# B&R Automation Studio project TD52 (part 127)

#### MeNoiAL.h
```c
/********************************************************************
 * COPYRIGHT -- Bernecker + Rainer Industrie-Elektronik Ges.m.b.H.
 ********************************************************************
 * Program: MeNoiAL
 * File: MeNoiAL.h
 * Author: 120011115
 * Created: Mon Sep 05 16:14:57 2016
 ********************************************************************
 * Header for program MeNoiAL
 ********************************************************************
 * Generated with B&R Automation Studio Target for Simulink V4.2
 * (ERT based)
 ********************************************************************/

#ifndef RTW_HEADER_MeNoiAL_h_
#define RTW_HEADER_MeNoiAL_h_
#ifndef MeNoiAL_COMMON_INCLUDES_
# define MeNoiAL_COMMON_INCLUDES_
#include <math.h>
#include "rtwtypes.h"
#endif                                 /* MeNoiAL_COMMON_INCLUDES_ */

#include "MeNoiAL_types.h"
#include "lMeNoiAL.h"

/* Macros for accessing real-time model data structure */
#ifndef rtmGetErrorStatus
# define rtmGetErrorStatus(rtm)        ((void*) 0)
#endif

#ifndef rtmSetErrorStatus
# define rtmSetErrorStatus(rtm, val)   ((void) 0)
#endif

#ifndef rtmGetStopRequested
# define rtmGetStopRequested(rtm)      ((void*) 0)
#endif

#ifndef MIN
#define MIN(a,b)                       ((a) < (b) ? (a) : (b))
#endif

#ifndef MAX
#define MAX(a,b)                       ((a) > (b) ? (a) : (b))
#endif

/* user code (top of header file) */
/***************************************************************************************************
 * COPYRIGHT -- INNIO Jenbacher GmbH & CO OG
 ****************************************************************************************************
 * Program:            MeNoiAL
 * Author:             schmisi00
 * Created:            12.03.2020 09:42
 ****************************************************************************************************
 * MODEL INFORMATION
 ****************************************************************************************************
 * Model Name:         C:\Git\ValveFractureMonitoring\KN_MechNoiseAdapLim\MeNoiAL.slx
 * Model Version:      1.03
 * Simulink Version:   R2012b
 * B&R Target:         V4.5.1
 * Description:        Mechanical Noise Monitoring Function.
 *
 *                     Outstandings:
 *                     -------------
 *                     - NA
 ****************************************************************************************************
 * HISTORY
 ****************************************************************************************************
 * Last Modified By:   schmisi00
 * Last Modified Date: Thu Mar 12 09:41:58 2020
 * Modified Comment:   V1.00 - 20.09.2019 - Created, model implementation from AS to Simulink
 *                     V1.01 - 11.11.2019 - Removed trigger (Para.bMeNoi_Active) from adaptive limit calculation block
 *                     V1.02 - 21.11.2019 - Model cleanup, removed parameter rFiltGain_MeNoi and rFiltOffsFac_MeNoi
 *                     V1.03 - 12.03.2020 - Fenst2_Min calculation change to avoid 65535 during engine standstill
 ****************************************************************************************************/

/* Block signals (auto storage) */

/* Block states (auto storage) for system '<Root>' */

/* Invariant block signals (auto storage) */

/* External inputs (root inport signals with auto storage) */

/* External outputs (root outports fed by signals with auto storage) */

extern const ConstBlockIO_MeNoiAL MeNoiAL_ConstB;/* constant block i/o */

/* Model entry point functions */
extern void MeNoiAL_initialize(D_Work_MeNoiAL *MeNoiAL_DWork, struct fMeNoiAL* inst);
extern void MeNoiAL_step(BlockIO_MeNoiAL *MeNoiAL_B, D_Work_MeNoiAL
  *MeNoiAL_DWork, ExternalOutputs_MeNoiAL *MeNoiAL_Y, struct fMeNoiAL* inst);
extern void MeNoiAL_terminate(struct fMeNoiAL* inst);

/*-
 * The generated code includes comments that allow you to trace directly
 * back to the appropriate location in the model.  The basic format
 * is <system>/block_name, where system is the system number (uniquely
 * assigned by Simulink) and block_name is the name of the block.
 *
 * Use the MATLAB hilite_system command to trace the generated code back
 * to the model.  For example,
 *
 * hilite_system('<S3>')    - opens system 3
 * hilite_system('<S3>/Kp') - opens and selects block Kp which resides in S3
 *
 * Here is the system hierarchy for this model
 *
 * '<Root>' : 'MeNoiAL'
 * '<S1>'   : 'MeNoiAL/Environment Controller'
 * '<S2>'   : 'MeNoiAL/Environment Controller1'
 * '<S3>'   : 'MeNoiAL/Fenst2 Thresh Alarm'
 * '<S4>'   : 'MeNoiAL/Fenst2_Average_Min_Max'
 * '<S5>'   : 'MeNoiAL/Info'
 * '<S6>'   : 'MeNoiAL/Mechanical Noise Adaptive Limit'
 * '<S7>'   : 'MeNoiAL/PARA_Limitation'
 * '<S8>'   : 'MeNoiAL/Fenst2_Average_Min_Max/Divisor'
 * '<S9>'   : 'MeNoiAL/Fenst2_Average_Min_Max/MATLAB Function1'
 * '<S10>'  : 'MeNoiAL/Fenst2_Average_Min_Max/Divisor/Data Type Conversion Inherited'
 * '<S11>'  : 'MeNoiAL/Mechanical Noise Adaptive Limit/Backward Euler PT1'
 * '<S12>'  : 'MeNoiAL/Mechanical Noise Adaptive Limit/Divisor'
 * '<S13>'  : 'MeNoiAL/Mechanical Noise Adaptive Limit/Saturation Dynamic'
 * '<S14>'  : 'MeNoiAL/Mechanical Noise Adaptive Limit/Saturation Dynamic1'
 * '<S15>'  : 'MeNoiAL/Mechanical Noise Adaptive Limit/Backward Euler PT1/Divisor'
 * '<S16>'  : 'MeNoiAL/Mechanical Noise Adaptive Limit/Backward Euler PT1/Divisor/Data Type Conversion Inherited'
 * '<S17>'  : 'MeNoiAL/Mechanical Noise Adaptive Limit/Divisor/Data Type Conversion Inherited'
 */
#endif                                 /* RTW_HEADER_MeNoiAL_h_ */
```

#### MeNoiAL_private.h
```c
/********************************************************************
 * COPYRIGHT -- Bernecker + Rainer Industrie-Elektronik Ges.m.b.H.
 ********************************************************************
 * Program: MeNoiAL
 * File: MeNoiAL_private.h
 * Author: 120011115
 * Created: Mon Sep 05 16:14:57 2016
 ********************************************************************
 * Header for program MeNoiAL
 ********************************************************************
 * Generated with B&R Automation Studio Target for Simulink V4.2
 * (ERT based)
 ********************************************************************/

#ifndef RTW_HEADER_MeNoiAL_private_h_
#define RTW_HEADER_MeNoiAL_private_h_
#include "rtwtypes.h"
#include <bur/plctypes.h>
#ifndef __RTWTYPES_H__
#error This file requires rtwtypes.h to be included
#else
#ifdef TMWTYPES_PREVIOUSLY_INCLUDED
#error This file requires rtwtypes.h to be included before tmwtypes.h
#else

/* Check for inclusion of an incorrect version of rtwtypes.h */
#ifndef RTWTYPES_ID_C08S16I32L32N32F1
#error This code was generated with a different "rtwtypes.h" than the file included
#endif                                 /* RTWTYPES_ID_C08S16I32L32N32F1 */
#endif                                 /* TMWTYPES_PREVIOUSLY_INCLUDED */
#endif                                 /* __RTWTYPES_H__ */

#ifndef MIN
#define MIN(a,b)                       ((a) < (b) ? (a) : (b))
#endif

#ifndef MAX
#define MAX(a,b)                       ((a) > (b) ? (a) : (b))
#endif
#endif                                 /* RTW_HEADER_MeNoiAL_private_h_ */
```

#### MeNoiAL_types.h
```c
/********************************************************************
 * COPYRIGHT -- Bernecker + Rainer Industrie-Elektronik Ges.m.b.H.
 ********************************************************************
 * Program: MeNoiAL
 * File: MeNoiAL_types.h
 * Author: 120011115
 * Created: Mon Sep 05 16:14:57 2016
 ********************************************************************
 * Header for program MeNoiAL
 ********************************************************************
 * Generated with B&R Automation Studio Target for Simulink V4.2
 * (ERT based)
 ********************************************************************/

#ifndef RTW_HEADER_MeNoiAL_types_h_
#define RTW_HEADER_MeNoiAL_types_h_
#include "rtwtypes.h"
#ifndef MIN
#define MIN(a,b)                       ((a) < (b) ? (a) : (b))
#endif

#ifndef MAX
#define MAX(a,b)                       ((a) > (b) ? (a) : (b))
#endif

#endif                                 /* RTW_HEADER_MeNoiAL_types_h_ */
```

#### rtwtypes.h
```c
/********************************************************************
 * COPYRIGHT -- Bernecker + Rainer Industrie-Elektronik Ges.m.b.H.
 ********************************************************************
 * Program: MeNoiAL
 * File: rtwtypes.h
 * Author: 120011115
 * Created: Mon Sep 05 16:14:57 2016
 ********************************************************************
 * Header for program MeNoiAL
 ********************************************************************
 * Generated with B&R Automation Studio Target for Simulink V4.2
 * (ERT based)
 ********************************************************************/

#ifndef __RTWTYPES_H__
#define __RTWTYPES_H__
#ifndef TRUE
# define TRUE                          (1U)
#endif

#ifndef FALSE
# define FALSE                         (0U)
#endif

#ifndef __TMWTYPES__
#define __TMWTYPES__
#include <limits.h>

/*=======================================================================*
 * Target hardware information
 *   Device type: Intel->x86/Pentium
 *   Number of bits:     char:   8    short:   16    long:  32
 *                       long:  32
 *                       native word size:  32
 *   Byte ordering: LittleEndian
 *   Signed integer division rounds to: Zero
 *   Shift right on a signed integer as arithmetic shift: on
 *=======================================================================*/

/*=======================================================================*
 * Fixed width word size data types:                                     *
 *   int8_T, int16_T, int32_T     - signed 8, 16, or 32 bit integers     *
 *   uint8_T, uint16_T, uint32_T  - unsigned 8, 16, or 32 bit integers   *
 *   real32_T, real64_T           - 32 and 64 bit floating point numbers *
 *=======================================================================*/
typedef signed char int8_T;
typedef unsigned char uint8_T;
typedef short int16_T;
typedef unsigned short uint16_T;
typedef long int32_T;
typedef unsigned long uint32_T;
typedef float real32_T;
typedef double real64_T;

/*===========================================================================*
 * Generic type definitions: real_T, time_T, boolean_T, int_T, uint_T,       *
 *                           ulong_T, char_T and byte_T.                     *
 *===========================================================================*/
typedef double real_T;
typedef double time_T;
typedef unsigned char boolean_T;
typedef long int_T;
typedef unsigned long uint_T;
typedef unsigned long ulong_T;
typedef char char_T;
typedef unsigned char uchar_T;
typedef char_T byte_T;

/*=======================================================================*
 * Min and Max:                                                          *
 *   int8_T, int16_T, int32_T     - signed 8, 16, or 32 bit integers     *
 *   uint8_T, uint16_T, uint32_T  - unsigned 8, 16, or 32 bit integers   *
 *=======================================================================*/
#define MAX_int8_T                     ((int8_T)(127))
#define MIN_int8_T                     ((int8_T)(-128))
#define MAX_uint8_T                    ((uint8_T)(255U))
#define MIN_uint8_T                    ((uint8_T)(0U))
#define MAX_int16_T                    ((int16_T)(32767))
#define MIN_int16_T                    ((int16_T)(-32768))
#define MAX_uint16_T                   ((uint16_T)(65535U))
#define MIN_uint16_T                   ((uint16_T)(0U))
#define MAX_int32_T                    ((int32_T)(2147483647))
#define MIN_int32_T                    ((int32_T)(-2147483647-1))
#define MAX_uint32_T                   ((uint32_T)(0xFFFFFFFFU))
#define MIN_uint32_T                   ((uint32_T)(0U))

/* Logical type definitions */
#if (!defined(__cplusplus)) && (!defined(__true_false_are_keywords))
#  ifndef false
#   define false                       (0U)
#  endif

#  ifndef true
#   define true                        (1U)
#  endif
#endif

/*
 * Simulink Coder assumes the code is compiled on a target using a 2's complement representation
 * for signed integer values.
 */
#if ((SCHAR_MIN + 1) != -SCHAR_MAX)
#error "This code must be compiled using a 2's complement representation for signed integer values"
#endif

/* This ID is used to detect inclusion of an incompatible rtwtypes.h */
#define RTWTYPES_ID_C08S16I32L32N32F1
#else                                  /* __TMWTYPES__ */
#define TMWTYPES_PREVIOUSLY_INCLUDED
#endif                                 /* __TMWTYPES__ */

/* Block D-Work pointer type */
typedef void * pointer_T;

/* Simulink specific types */
#ifndef __SIMSTRUC_TYPES_H__
#define __SIMSTRUC_TYPES_H__

/* Trigger directions: falling, either, and rising */
typedef enum {
  FALLING_ZERO_CROSSING = -1,
  ANY_ZERO_CROSSING = 0,
  RISING_ZERO_CROSSING = 1
} ZCDirection;

/* Previous state of a trigger signal */
typedef uint8_T ZCSigState;

/* Initial value of a trigger zero crossing signal */
#define UNINITIALIZED_ZCSIG            0x03U
#define NEG_ZCSIG                      0x02U
#define POS_ZCSIG                      0x01U
#define ZERO_ZCSIG                     0x00U

/* Current state of a trigger signal */
typedef enum {
  FALLING_ZCEVENT = -1,
  NO_ZCEVENT = 0,
  RISING_ZCEVENT = 1
} ZCEventType;

#endif                                 /* __SIMSTRUC_TYPES_H__ */
#endif                                 /* __RTWTYPES_H__ */

#ifndef MIN
#define MIN(a,b)                       ((a) < (b) ? (a) : (b))
#endif

#ifndef MAX
#define MAX(a,b)                       ((a) > (b) ? (a) : (b))
#endif
```

#### MeNoiAL.c
```c
/********************************************************************
 * COPYRIGHT -- Bernecker + Rainer Industrie-Elektronik Ges.m.b.H.
 ********************************************************************
 * Program: MeNoiAL
 * File: MeNoiAL.c
 * Author: 120011115
 * Created: Mon Sep 05 16:14:57 2016
 ********************************************************************
 * Implementation of program MeNoiAL
 ********************************************************************
 * Generated with B&R Automation Studio Target for Simulink V4.2
 * (ERT based)
 ********************************************************************/
#include "MeNoiAL.h"
#include "MeNoiAL_private.h"

/*  Defines */

/*  Data Types */

/**************************** GLOBAL DATA *************************************/
/*  Definitions */

/*  Declarations  */

/***************************** FILE SCOPE DATA ********************************/

/*************************** FUNCTIONS ****************************************/

/* Model step function */
void MeNoiAL_step(struct BlockIO_MeNoiAL *MeNoiAL_B, struct D_Work_MeNoiAL *MeNoiAL_DWork,
                  ExternalOutputs_MeNoiAL *MeNoiAL_Y, struct fMeNoiAL* inst)
{
  /* local block i/o variables */
  boolean_T rtb_LogicalOperator;
  real32_T rtb_rFiltTau_MeNoi;
  real32_T rtb_rMargTExh_Active;
  real32_T rtb_rFenst2LiMn;
  real32_T rtb_Switch4;
  real32_T rtb_Divide;
  uint16_T rtb_Divide1[25];
  real32_T rtb_Switch;
  real32_T rtb_Switch3;
  real32_T rtb_Switch5;
  boolean_T rtb_y[25];
  real32_T rtb_Switch2_h[25];
  int32_T i;
  uint8_T rtb_SumofElements1;
  uint32_T tmp;
  boolean_T rtb_RelationalOperator_m;
  real32_T rtb_SumofElements_k;
  real32_T DiscreteTimeIntegrator[25];
  int32_T i_0;
  int32_T i_1;
  int16_T e_data[25];
  int16_T tmp_data[25];
  boolean_T rtb_LowerRelop;
  real32_T DiscreteTimeIntegrator_0;
  int32_T i_2;

  /* S-Function (bur_bus_in): '<Root>/Bus Input1' */
  MeNoiAL_B->BusInput1 = inst->Para;

  /* BusSelector: '<Root>/Bus Selector6' */
  rtb_rFiltTau_MeNoi = MeNoiAL_B->BusInput1.rFiltTau_MeNoi;
  rtb_rMargTExh_Active = MeNoiAL_B->BusInput1.rMargTExh_Active;
  rtb_rFenst2LiMn = MeNoiAL_B->BusInput1.rFenst2LiMn;

  /* Switch: '<S7>/Switch4' incorporates:
   *  BusSelector: '<Root>/Bus Selector6'
   *  Constant: '<S7>/Constant4'
   */
  if (MeNoiAL_B->BusInput1.rFenst2LiMx != 0.0F) {
    /* Saturate: '<S7>/Saturation4' */
    if (MeNoiAL_B->BusInput1.rFenst2LiMx >= 16000.0F) {
      rtb_Switch4 = 16000.0F;
    } else if (MeNoiAL_B->BusInput1.rFenst2LiMx <= 0.0F) {
      rtb_Switch4 = 0.0F;
    } else {
      rtb_Switch4 = MeNoiAL_B->BusInput1.rFenst2LiMx;
    }

    /* End of Saturate: '<S7>/Saturation4' */
  } else {
    rtb_Switch4 = 2000.0F;
  }

  /* End of Switch: '<S7>/Switch4' */

  /* S-Function (bur_bus_in): '<Root>/Bus Input' */
  MeNoiAL_B->BusInput = inst->In;

  /* Switch: '<S7>/Switch5' incorporates:
   *  Constant: '<S7>/Constant5'
   */
  if (rtb_rFenst2LiMn != 0.0F) {
    /* Saturate: '<S7>/Saturation5' */
    if (rtb_rFenst2LiMn >= 16000.0F) {
      rtb_Switch5 = 16000.0F;
    } else if (rtb_rFenst2LiMn <= 0.0F) {
      rtb_Switch5 = 0.0F;
    } else {
      rtb_Switch5 = rtb_rFenst2LiMn;
    }

    /* End of Saturate: '<S7>/Saturation5' */
  } else {
    rtb_Switch5 = 30.0F;
  }

  /* End of Switch: '<S7>/Switch5' */

  /* Switch: '<S7>/Switch' incorporates:
   *  Constant: '<S7>/Constant'
   */
  if (rtb_rFiltTau_MeNoi != 0.0F) {
    /* Saturate: '<S7>/Saturation' */
    if (rtb_rFiltTau_MeNoi >= 50.0F) {
      rtb_Switch = 50.0F;
    } else if (rtb_rFiltTau_MeNoi <= 0.0F) {
      rtb_Switch = 0.0F;
    } else {
      rtb_Switch = rtb_rFiltTau_MeNoi;
    }

    /* End of Saturate: '<S7>/Saturation' */
  } else {
    rtb_Switch = 5.0F;
  }

  /* End of Switch: '<S7>/Switch' */

  /* Product: '<S7>/Divide' incorporates:
   *  Constant: '<S7>/Constant2'
   */
  rtb_Divide = rtb_Switch4 / 3.5F;

  /* Switch: '<S7>/Switch3' incorporates:
   *  Constant: '<S7>/Constant3'
   */
  if (rtb_rMargTExh_Active != 0.0F) {
    /* Saturate: '<S7>/Saturation3' */
    if (rtb_rMargTExh_Active >= 1.0F) {
      rtb_Switch3 = 1.0F;
    } else if (rtb_rMargTExh_Active <= 0.0F) {
      rtb_Switch3 = 0.0F;
    } else {
      rtb_Switch3 = rtb_rMargTExh_Active;
    }

    /* End of Saturate: '<S7>/Saturation3' */
  } else {
    rtb_Switch3 = 0.15F;
  }

  /* End of Switch: '<S7>/Switch3' */

  /* Outputs for Atomic SubSystem: '<Root>/Fenst2_Average_Min_Max' */
  /* MATLAB Function: '<S4>/MATLAB Function1' */
  /* MATLAB Function 'Fenst2_Average_Min_Max/MATLAB Function1': '<S9>:1' */
  /* '<S9>:1:3' */
  for (i_0 = 0; i_0 < 25; i_0++) {
    rtb_y[i_0] = FALSE;
  }

  i_2 = (int32_T)((uint32_T)MeNoiAL_B->BusInput.ucNumCyl + 1U);
  if ((uint32_T)i_2 > 255U) {
    i_2 = 255;
  }

  if (2 > (uint8_T)i_2) {
    i = 1;
    i_2 = 0;
  } else {
    i = 2;
    i_2 = (uint8_T)i_2;
  }

  i_0 = i_2 - i;
  for (i_1 = 0; i_1 <= i_0; i_1++) {
    tmp_data[i_1] = (int16_T)(i + i_1);
  }

  i_0 = (i_2 - i) + 1;
  for (i_2 = 0; i_2 < i_0; i_2++) {
    for (i = 0; i < 1; i++) {
      e_data[i_2] = tmp_data[i_2];
    }
  }

  /* '<S9>:1:4' */
  for (i_2 = 0; i_2 < i_0; i_2++) {
    rtb_y[e_data[i_2] - 1] = TRUE;
  }

  /* output */
  /* '<S9>:1:7' */
  for (i_2 = 0; i_2 < 25; i_2++) {
    /* Logic: '<S4>/Logical Operator' incorporates:
     *  Logic: '<S4>/Logical Operator2'
     *  Product: '<S4>/Divide1'
     */
    rtb_RelationalOperator_m = (rtb_y[i_2] && (!MeNoiAL_B->
      BusInput.bKnockSig[i_2]));

    /* Product: '<S4>/Divide1' incorporates:
     *  DataTypeConversion: '<S4>/Data Type Conversion5'
     */
    rtb_Divide1[i_2] = (uint16_T)(rtb_RelationalOperator_m ?
      MeNoiAL_B->BusInput.uFenst2[i_2] : 0);

    /* Logic: '<S4>/Logical Operator' */
    rtb_y[i_2] = rtb_RelationalOperator_m;
  }

  /* End of MATLAB Function: '<S4>/MATLAB Function1' */

  /* Sum: '<S4>/Sum of Elements1' */
  tmp = (uint32_T)rtb_y[0];
  for (i_2 = 0; i_2 < 24; i_2++) {
    tmp += (uint32_T)rtb_y[i_2 + 1];
  }

  rtb_SumofElements1 = (uint8_T)tmp;

  /* End of Sum: '<S4>/Sum of Elements1' */

  /* Switch: '<S4>/Switch' incorporates:
   *  Constant: '<S4>/Constant2'
   *  DataTypeConversion: '<S4>/Data Type Conversion4'
   *  Product: '<S4>/Divide'
   */
  if (rtb_SumofElements1 != 0) {
    /* Sum: '<S4>/Sum of Elements' */
    rtb_SumofElements_k = (real32_T)rtb_Divide1[0];
    for (i_2 = 0; i_2 < 24; i_2++) {
      rtb_SumofElements_k += (real32_T)rtb_Divide1[i_2 + 1];
    }

    /* End of Sum: '<S4>/Sum of Elements' */

    /* Switch: '<S8>/Switch' incorporates:
     *  RelationalOperator: '<S8>/Relational Operator'
     */
    if (1 >= rtb_SumofElements1) {
      rtb_SumofElements1 = 1U;
    }

    /* End of Switch: '<S8>/Switch' */
    rtb_rFiltTau_MeNoi = rtb_SumofElements_k / (real32_T)rtb_SumofElements1;
  } else {
    rtb_rFiltTau_MeNoi = 0.0F;
  }

  /* End of Switch: '<S4>/Switch' */

  /* MinMax: '<S4>/MinMax1' */
  rtb_rMargTExh_Active = (real32_T)rtb_Divide1[0];
  for (i = 0; i < 24; i++) {
    if (!(rtb_rMargTExh_Active >= (real32_T)rtb_Divide1[i + 1])) {
      rtb_rMargTExh_Active = (real32_T)rtb_Divide1[i + 1];
    }
  }

  /* Switch: '<S4>/Switch2' incorporates:
   *  Constant: '<S4>/Constant3'
   */
  for (i_0 = 0; i_0 < 25; i_0++) {
    if (rtb_y[i_0]) {
      rtb_Switch2_h[i_0] = (real32_T)rtb_Divide1[i_0];
    } else {
      rtb_Switch2_h[i_0] = 65535.0F;
    }
  }

  /* End of Switch: '<S4>/Switch2' */

  /* MinMax: '<S4>/MinMax' */
  rtb_SumofElements_k = rtb_Switch2_h[0];
  for (i = 0; i < 24; i++) {
    if (!(rtb_SumofElements_k <= rtb_Switch2_h[i + 1])) {
      rtb_SumofElements_k = rtb_Switch2_h[i + 1];
    }
  }

  /* End of Outputs for SubSystem: '<Root>/Fenst2_Average_Min_Max' */

  /* Outputs for Atomic SubSystem: '<Root>/Mechanical Noise Adaptive Limit' */
  /* DataTypeConversion: '<S6>/Data Type Conversion1' */
  for (i_0 = 0; i_0 < 25; i_0++) {
    rtb_Switch2_h[i_0] = (real32_T)MeNoiAL_B->BusInput.uFenst2[i_0];
  }

  /* End of DataTypeConversion: '<S6>/Data Type Conversion1' */

  /* Outputs for Atomic SubSystem: '<S6>/Backward Euler PT1' */
  /* Switch: '<S15>/Switch' incorporates:
   *  Abs: '<S15>/Abs'
   *  RelationalOperator: '<S15>/Relational Operator'
   */
  if (2.22044605E-16F >= rtb_Switch) {
    rtb_rFenst2LiMn = 2.22044605E-16F;
  } else {
    rtb_rFenst2LiMn = rtb_Switch;
  }

  /* End of Switch: '<S15>/Switch' */

  /* RelationalOperator: '<S11>/Relational Operator' incorporates:
   *  Constant: '<S11>/Constant'
   */
  rtb_RelationalOperator_m = (rtb_Switch > 0.0F);

  /* Logic: '<S11>/Logical Operator' incorporates:
   *  Logic: '<S11>/Logical Operator1'
   */
  rtb_LogicalOperator = !rtb_RelationalOperator_m;

  /* DiscreteIntegrator: '<S11>/Discrete-Time Integrator' */
  if (MeNoiAL_DWork->DiscreteTimeIntegrator_IC_LOADI != 0) {
    for (i_0 = 0; i_0 < 25; i_0++) {
      MeNoiAL_DWork->DiscreteTimeIntegrator_DSTATE[i_0] = rtb_Switch2_h[i_0];
    }
  }

  /* Update for DiscreteIntegrator: '<S11>/Discrete-Time Integrator' */
  MeNoiAL_DWork->DiscreteTimeIntegrator_IC_LOADI = 0U;
  for (i_0 = 0; i_0 < 25; i_0++) {
    /* DiscreteIntegrator: '<S11>/Discrete-Time Integrator' incorporates:
     *  Delay: '<S11>/Delay'
     *  Product: '<S11>/Divide4'
     *  Sum: '<S11>/Sum4'
     */
    if (rtb_LogicalOperator || (MeNoiAL_DWork->DiscreteTimeIntegrator_PrevRese
         != 0)) {
      MeNoiAL_DWork->DiscreteTimeIntegrator_DSTATE[i_0] = rtb_Switch2_h[i_0];
    }

    DiscreteTimeIntegrator_0 = (rtb_Switch2_h[i_0] - MeNoiAL_DWork->
      Delay_DSTATE[i_0]) / rtb_rFenst2LiMn * 0.01F +
      MeNoiAL_DWork->DiscreteTimeIntegrator_DSTATE[i_0];

    /* Update for Delay: '<S11>/Delay' */
    MeNoiAL_DWork->Delay_DSTATE[i_0] = DiscreteTimeIntegrator_0;

    /* Update for DiscreteIntegrator: '<S11>/Discrete-Time Integrator' */
    MeNoiAL_DWork->DiscreteTimeIntegrator_DSTATE[i_0] = DiscreteTimeIntegrator_0;

    /* Sum: '<S6>/Add2' incorporates:
     *  Constant: '<S6>/Constant3'
     *  Product: '<S6>/Product1'
     *  Switch: '<S11>/Switch'
     */
    if (!rtb_RelationalOperator_m) {
      DiscreteTimeIntegrator_0 = rtb_Switch2_h[i_0];
    }

    DiscreteTimeIntegrator_0 = DiscreteTimeIntegrator_0 * 1.1F + rtb_Divide;

    /* End of Sum: '<S6>/Add2' */

    /* RelationalOperator: '<S13>/LowerRelop1' */
    rtb_LowerRelop = (DiscreteTimeIntegrator_0 > rtb_Switch4);

    /* Switch: '<S13>/Switch' incorporates:
     *  RelationalOperator: '<S13>/UpperRelop'
     */
    if (DiscreteTimeIntegrator_0 < rtb_Switch5) {
      DiscreteTimeIntegrator_0 = rtb_Switch5;
    }

    /* End of Switch: '<S13>/Switch' */

    /* Switch: '<S13>/Switch2' */
    if (rtb_LowerRelop) {
      DiscreteTimeIntegrator_0 = rtb_Switch4;
    }

    /* End of Switch: '<S13>/Switch2' */

    /* Product: '<S6>/Divide2' */
    DiscreteTimeIntegrator_0 = rtb_y[i_0] ? DiscreteTimeIntegrator_0 : 0.0F;
    DiscreteTimeIntegrator[i_0] = DiscreteTimeIntegrator_0;
  }

  /* Update for DiscreteIntegrator: '<S11>/Discrete-Time Integrator' */
  if (rtb_LogicalOperator) {
    MeNoiAL_DWork->DiscreteTimeIntegrator_PrevRese = 1;
  } else {
    MeNoiAL_DWork->DiscreteTimeIntegrator_PrevRese = 0;
  }

  /* End of Outputs for SubSystem: '<S6>/Backward Euler PT1' */

  /* Sum: '<S6>/Sum of Elements1' */
  tmp = (uint32_T)rtb_y[0];
  for (i_2 = 0; i_2 < 24; i_2++) {
    tmp += (uint32_T)rtb_y[i_2 + 1];
  }

  rtb_SumofElements1 = (uint8_T)tmp;

  /* End of Sum: '<S6>/Sum of Elements1' */

  /* Switch: '<S6>/Switch' incorporates:
   *  Constant: '<S6>/Constant2'
   *  DataTypeConversion: '<S6>/Data Type Conversion6'
   *  Product: '<S6>/Divide'
   */
  if (rtb_SumofElements1 != 0) {
    /* Sum: '<S6>/Sum of Elements' */
    rtb_rFenst2LiMn = DiscreteTimeIntegrator[0];
    for (i_2 = 0; i_2 < 24; i_2++) {
      rtb_rFenst2LiMn += DiscreteTimeIntegrator[i_2 + 1];
    }

    /* End of Sum: '<S6>/Sum of Elements' */

    /* Switch: '<S12>/Switch' incorporates:
     *  Constant: '<S12>/Constant2'
     *  RelationalOperator: '<S12>/Relational Operator'
     */
    if (1 >= rtb_SumofElements1) {
      i_2 = 1;
    } else {
      i_2 = rtb_SumofElements1;
    }

    /* End of Switch: '<S12>/Switch' */
    rtb_rFenst2LiMn /= (real32_T)i_2;
  } else {
    rtb_rFenst2LiMn = 0.0F;
  }

  /* End of Switch: '<S6>/Switch' */

  /* Sum: '<S6>/Add1' incorporates:
   *  Product: '<S6>/Product2'
   */
  rtb_rFenst2LiMn += rtb_Switch4 * rtb_Switch3;

  /* Switch: '<S14>/Switch2' incorporates:
   *  RelationalOperator: '<S14>/LowerRelop1'
   *  RelationalOperator: '<S14>/UpperRelop'
   *  Switch: '<S14>/Switch'
   */
  if (rtb_rFenst2LiMn > rtb_Switch4) {
    rtb_rFenst2LiMn = rtb_Switch4;
  } else {
    if (rtb_rFenst2LiMn < rtb_Switch5) {
      /* Switch: '<S14>/Switch' */
      rtb_rFenst2LiMn = rtb_Switch5;
    }
  }

  /* End of Switch: '<S14>/Switch2' */
  /* End of Outputs for SubSystem: '<Root>/Mechanical Noise Adaptive Limit' */

  /* Outputs for Atomic SubSystem: '<Root>/Fenst2 Thresh Alarm' */
  /* Switch: '<S3>/Switch' incorporates:
   *  Product: '<S3>/Product'
   */
  if (MeNoiAL_B->BusInput1.bMeNoi_Active) {
    for (i_0 = 0; i_0 < 25; i_0++) {
      rtb_Switch2_h[i_0] = DiscreteTimeIntegrator[i_0];
    }
  } else {
    for (i_0 = 0; i_0 < 25; i_0++) {
      rtb_Switch2_h[i_0] = rtb_Switch4 * MeNoiAL_ConstB.DataTypeConversion[i_0];
    }
  }

  for (i_0 = 0; i_0 < 25; i_0++) {
    /* RelationalOperator: '<S3>/Relational Operator' */
    rtb_LowerRelop = ((real32_T)rtb_Divide1[i_0] > rtb_Switch2_h[i_0]);

    /* Switch: '<S3>/Switch1' incorporates:
     *  Constant: '<S3>/Constant'
     *  Constant: '<S3>/Constant1'
     *  Delay: '<S3>/Delay'
     *  Sum: '<S3>/Sum'
     */
    if (rtb_LowerRelop) {
      rtb_SumofElements1 = (uint8_T)((uint32_T)MeNoiAL_DWork->Delay_DSTATE_c[i_0]
        + 1U);
    } else {
      rtb_SumofElements1 = 0U;
    }

    /* End of Switch: '<S3>/Switch1' */

    /* Logic: '<S3>/ 1' incorporates:
     *  Constant: '<S3>/Constant2'
     *  RelationalOperator: '<S3>/Relational Operator1'
     */
    rtb_RelationalOperator_m = ((rtb_SumofElements1 > 150) &&
      MeNoiAL_B->BusInput.bGCB_On_TC2_Di);

    /* Switch: '<S3>/Switch2' incorporates:
     *  Constant: '<S3>/Constant3'
     */
    if (rtb_RelationalOperator_m) {
      rtb_SumofElements1 = 150U;
    }

    /* End of Switch: '<S3>/Switch2' */

    /* Update for Delay: '<S3>/Delay' */
    MeNoiAL_DWork->Delay_DSTATE_c[i_0] = rtb_SumofElements1;

    /* BusCreator: '<Root>/Bus Creator' incorporates:
     *  Logic: '<S3>/ '
     *  Logic: '<S3>/ 2'
     *  Logic: '<S3>/Logical Operator'
     *  RelationalOperator: '<S3>/Relational Operator2'
     */
    MeNoiAL_Y->Out_MeNoiAL.bTExh_Mon_UseNarrowWindow[i_0] =
      ((MeNoiAL_B->BusInput1.bMeNoi_Active && rtb_LowerRelop) ||
       (MeNoiAL_B->BusInput1.bMeNoi_Active && (DiscreteTimeIntegrator[i_0] >
         rtb_rFenst2LiMn)));
    MeNoiAL_Y->Out_MeNoiAL.bValve[i_0] = rtb_RelationalOperator_m;

    /* BusCreator: '<Root>/Bus Creator1' */
    MeNoiAL_Y->Dbg_MeNoiAL.uMeNoi_Cnt[i_0] = rtb_SumofElements1;
    MeNoiAL_Y->Dbg_MeNoiAL.rFenst2_Vect[i_0] = (real32_T)rtb_Divide1[i_0];
    MeNoiAL_Y->Dbg_MeNoiAL.bValidCyl[i_0] = rtb_y[i_0];
  }

  /* End of Switch: '<S3>/Switch' */
  /* End of Outputs for SubSystem: '<Root>/Fenst2 Thresh Alarm' */

  /* Outputs for Atomic SubSystem: '<Root>/Fenst2_Average_Min_Max' */
  /* BusCreator: '<Root>/Bus Creator' incorporates:
   *  DataTypeConversion: '<S4>/Data Type Conversion1'
   *  DataTypeConversion: '<S4>/Data Type Conversion2'
   *  DataTypeConversion: '<S4>/Data Type Conversion3'
   *  MinMax: '<S4>/MinMax'
   *  MinMax: '<S4>/MinMax1'
   */
  MeNoiAL_Y->Out_MeNoiAL.uFenst2_Av = (uint16_T)(real32_T)fmod((real32_T)floor
    (rtb_rFiltTau_MeNoi), 65536.0F);
  MeNoiAL_Y->Out_MeNoiAL.uFenst2_Mx = (uint16_T)(int32_T)(real32_T)fmod
    (rtb_rMargTExh_Active, 65536.0F);
  MeNoiAL_Y->Out_MeNoiAL.uFenst2_Mn = (uint16_T)(int32_T)(real32_T)fmod
    (rtb_SumofElements_k, 65536.0F);

  /* End of Outputs for SubSystem: '<Root>/Fenst2_Average_Min_Max' */

  /* BusCreator: '<Root>/Bus Creator1' */
  MeNoiAL_Y->Dbg_MeNoiAL.rFiltTau_Lim = rtb_Switch;
  MeNoiAL_Y->Dbg_MeNoiAL.rFiltGain_Lim = 0.0F;
  MeNoiAL_Y->Dbg_MeNoiAL.rMargTexhAct_Lim = rtb_Switch3;
  MeNoiAL_Y->Dbg_MeNoiAL.rOffMeNoi_Lim = rtb_Divide;
  MeNoiAL_Y->Dbg_MeNoiAL.rFenst2LiMx_Lim = rtb_Switch4;
  MeNoiAL_Y->Dbg_MeNoiAL.rFenst2LiMn_Lim = rtb_Switch5;
  for (i_0 = 0; i_0 < 25; i_0++) {
    MeNoiAL_Y->Dbg_MeNoiAL.uAdapLim_MeNoi_Cyl[i_0] = DiscreteTimeIntegrator[i_0];
  }

  MeNoiAL_Y->Dbg_MeNoiAL.uAdapLim_Marg = rtb_rFenst2LiMn;

  /* S-Function (bur_bus_out): '<Root>/Bus Output' */
  inst->Out = MeNoiAL_Y->Out_MeNoiAL;

  /* S-Function (bur_bus_out): '<Root>/Bus Output1' */
  inst->Dbg = MeNoiAL_Y->Dbg_MeNoiAL;

  /* UnitDelay: '<S5>/Unit Delay' */
  MeNoiAL_B->UnitDelay = MeNoiAL_DWork->UnitDelay_DSTATE;

  /* S-Function (bur_out): '<Root>/Output' */
  inst->Version = MeNoiAL_B->UnitDelay;

  /* Update for UnitDelay: '<S5>/Unit Delay' */
  MeNoiAL_DWork->UnitDelay_DSTATE = 103U;
}

/* Model initialize function */
void MeNoiAL_initialize(struct D_Work_MeNoiAL *MeNoiAL_DWork, struct fMeNoiAL* inst)
{
  /* InitializeConditions for Atomic SubSystem: '<Root>/Mechanical Noise Adaptive Limit' */
  /* InitializeConditions for Atomic SubSystem: '<S6>/Backward Euler PT1' */
  /* InitializeConditions for DiscreteIntegrator: '<S11>/Discrete-Time Integrator' */
  MeNoiAL_DWork->DiscreteTimeIntegrator_IC_LOADI = 1U;

  /* End of InitializeConditions for SubSystem: '<S6>/Backward Euler PT1' */
  /* End of InitializeConditions for SubSystem: '<Root>/Mechanical Noise Adaptive Limit' */
}

/* Model terminate function */
void MeNoiAL_terminate(struct fMeNoiAL* inst)
{
  /* (no terminate code required) */
}

/*======================== TOOL VERSION INFORMATION ==========================*
 * MATLAB 8.0 (R2012b)20-Jul-2012                                             *
 * Simulink 8.0 (R2012b)20-Jul-2012                                           *
 * Simulink Coder 8.3 (R2012b)20-Jul-2012                                     *
 * Embedded Coder 6.3 (R2012b)20-Jul-2012                                     *
 * Stateflow 8.0 (R2012b)20-Jul-2012                                          *
 *============================================================================*/

/*======================= LICENSE IN USE INFORMATION =========================*
 * matlab                                                                     *
 * matlab_coder                                                               *
 * real-time_workshop                                                         *
 * rtw_embedded_coder                                                         *
 * simulink                                                                   *
 *============================================================================*/
```

#### MeNoiAL_data.c
```c
/********************************************************************
 * COPYRIGHT -- Bernecker + Rainer Industrie-Elektronik Ges.m.b.H.
 ********************************************************************
 * Program: MeNoiAL
 * File: MeNoiAL_data.c
 * Author: 120011115
 * Created: Mon Sep 05 16:14:57 2016
 ********************************************************************
 * Data for program MeNoiAL
 ********************************************************************
 * Generated with B&R Automation Studio Target for Simulink V4.2
 * (ERT based)
 ********************************************************************/
#include "MeNoiAL.h"
#include "MeNoiAL_private.h"

/*  GLOBAL DATA DEFINITIONS */

/* Invariant block signals (auto storage) */
const ConstBlockIO_MeNoiAL MeNoiAL_ConstB = {
  { 1.0F, 1.0F, 1.0F, 1.0F, 1.0F, 1.0F, 1.0F, 1.0F, 1.0F, 1.0F, 1.0F, 1.0F, 1.0F,
    1.0F, 1.0F, 1.0F, 1.0F, 1.0F, 1.0F, 1.0F, 1.0F, 1.0F, 1.0F, 1.0F, 1.0F }
  /* '<S3>/Data Type Conversion' */
};
```

#### fMeNoiAL.c
```c
/********************************************************************
 * COPYRIGHT -- Bernecker + Rainer Industrie-Elektronik Ges.m.b.H.
 ********************************************************************
 * Program: MeNoiAL
 * File: fMeNoiAL.c
 * Author: 120011115
 * Created: Mon Sep 05 16:14:57 2016
 ********************************************************************
 * Implementation of program MeNoiAL
 ********************************************************************
 * Generated with B&R Automation Studio Target for Simulink V4.2
 * (ERT based)
 ********************************************************************/
#include <bur/plctypes.h>
#include "MeNoiAL.h"
#include "rtwtypes.h"

/* Defines */
#define SS_TERMINATE 4
#define SS_OUTPUT 3
#define SS_INITIALIZE 2

/*  Data Types */

/**************************** GLOBAL DATA *************************************/
/*  Definitions */

/*  Declarations  */

/***************************** FILE SCOPE DATA ********************************/

/*************************** FUNCTIONS ****************************************/
#ifdef __cplusplus

unsigned long bur_heap_size = 6553500;

#endif

void fMeNoiAL(struct fMeNoiAL* inst)
{
  BlockIO_MeNoiAL *MeNoiAL_B = &(inst)->bur_BlockIO_MeNoiAL;
	D_Work_MeNoiAL *MeNoiAL_DWork = &(inst)->bur_D_Work_MeNoiAL;
	ExternalOutputs_MeNoiAL *MeNoiAL_Y = &(inst)->bur_ExternalOutputs_MeNoiAL;

  switch (inst->ssMethodType)
  {
   case SS_INITIALIZE:
    /* call model initialize function */
    MeNoiAL_initialize(MeNoiAL_DWork, inst);
    break;

   case SS_OUTPUT:
    /* call model step function */
    MeNoiAL_step(MeNoiAL_B, MeNoiAL_DWork, MeNoiAL_Y, inst);

    break;

   case SS_TERMINATE:
    /* call model terminate function */
    MeNoiAL_terminate(inst);
    break;
  }
}

/*****************************************************************************
   Function block sample time: 0.01s
 *****************************************************************************/

/*****************************************************************************
   B&R Automation Studio Target for Simulink Version: A4.5.1 (27-Jul-2015)
 *****************************************************************************/

/*======================== TOOL VERSION INFORMATION ==========================*
 * MATLAB 8.0 (R2012b)20-Jul-2012                                             *
 * Simulink 8.0 (R2012b)20-Jul-2012                                           *
 * Simulink Coder 8.3 (R2012b)20-Jul-2012                                     *
 * Embedded Coder 6.3 (R2012b)20-Jul-2012                                     *
 * Stateflow 8.0 (R2012b)20-Jul-2012                                          *
 *============================================================================*/

/*======================= LICENSE IN USE INFORMATION =========================*
 * matlab                                                                     *
 * matlab_coder                                                               *
 * real-time_workshop                                                         *
 * rtw_embedded_coder                                                         *
 * simulink                                                                   *
 *============================================================================*/
```

#### lib_properties.txt
```
For manual assignment to hardware configuration please
add the following additional include directories:

\Logical\MATLAB_includes\R2012b\

And the following additional build options:

-lm -D MODEL=MeNoiAL -D NUMST=1 -D NCSTATES=0 -D HAVESTDIO -D ONESTEPFCN=1 -D TERMFCN=1 -D MAT_FILE=0 -D MULTI_INSTANCE_CODE=1 -D INTEGER_CODE=0 -D MT=0 -D CLASSIC_INTERFACE=0 -D TID01EQ=0
```

### Data object Logical/Knocking/META_KN (Simple) - MODUL META data file

#### META_KN.dat
```
; *******************************************************************************
; AGGR: Module Meta Data (data module)
;
; This code is confidential and proprietary to the INNIO Company.
; It may not be used in any form, or reproduced in any manner, without the express
; written permission of the INNIO Company.
; Copyright, INNIO Company, 2025
;
; Customized modifications: -
; ------------------------
;
; History:
; -------
; V3.99			06-03-2013	Weitzer, 	generated for modular software
; V4.00 		31.01.2014	Weitzer, 	versions changed
; V4.01.00.00 	23.07.2014	Waldhart,	new interfaces added
; V4.02.00.00	16.02.2015	Caks,		added safi dmr
; V4.03.00.00	02.11.2015	Zengerer	add MANDATORYMODULE statement
; V4.04.00.00   18.04.2016	Gwiggner,   Bugfix ITP Interpolation GAS1-2
; V4.04.00.00	12.05.2016	502423184	versions changed,  SAFI_DMR Task for Type9 / G2
; V4.04.00.00	14.11.2016	Gwiggner	Bugfix: VISU knocking IP reduction
; V4.04.00.00   xx.03.2017	Farre,		Bugfix: adaptive knock limit safi_kls
; V4.04.00.00   15.05.2017	Gwiggner,	Bugfix: KLS98 validation - MSF not working
; V4.05.00.00   05.03.2018	Perktold,	Delaytime for MSF SAFI/KLS corrected 2.5sec instead of 0.3s, Type 6 "BlockAfterKnockTrip"
; V4.05.01.00   16.04.2018	Perktold,	Integrated comments regarding "Safety-related application software source code (EN 13849-1 / 4.6.3)"
; V4.06.00.00   28.09.2018	Gwiggner,	change A3342 Knock sensor measuring sensor failure from Prio 3 to Prio 2"
; V4.07.00.00	13.05.2019	Hohensinner	Added RKS Package
; V4.07.00.00	23.10.2019	Farre,		BU 01: avoiding division by 0
; V4.09.00.00	23.01.2020	Schmidt,	Mechanical noise monitoring for valve fracture detection added
; V4.10.00.00	19.01.2020	Farre,		added individual knocking threshold per Bank
; V4.10.00.00	28.01.2021	Denk,		Alarm deactivation when DGS/WinMOD Simulation is active (2438, 2439, 2440, 2441).
; V4.11.00.00	22.12.2021	Andre		Moved W2493 and B2939 to SAFI module. Added notification of frozen or knock noise from SAFI module.
; V4.11.00.00	14.01.2022	Schmidt		Changed bKnockSig variable to global (used for PU scuffing detection)
; V4.12.00.00	03.10.2022	Farre,		Issue #438: Current knock integrator value connected to AVG, MAX & MIN MM2VIS for KLS90
; 				03.10.2022	Farre,		Issue #906: J208 KLS90 uses only one knock sensor, second sensor is looped through
;				22.11.2022	Farre,		Feature: Introduction knock adaptive limit for Type4 with DMR
;				19.12.2022	Perktold	added comments for sr-code (EN 13849-1 / 4.6.3) for A3342
; V04.13.00.00	05.12.2023	Bencze		A1048,3339,3342: risc class 10 (for T6), no remote reset possible
; V04.14.00.00	19.07.2024	Kafka,		Remove G2 and add KLS as RKS system for T9
;							Andre,		Fix issue 1585.
;				21.01.2025	Gwiggner,	J208F KLS90 use of 2nd knock senor (#1791)
;
; Instructions for use:
; --------------------
; make only changes at the version numbers
;
; Outstandings:
; ------------
;
; *******************************************************************************
;
"<META>"
;
; Module ID
"<MODUL>KN</MODUL>"
;
; Module Version (xx.yy.zz.cc)
"<VERSION>04.14.00.00</VERSION>"
;
; Module Basisupdate Version BU (00-99)
"<BASISUPDATE_VERSION>00</BASISUPDATE_VERSION>"
;
; Optional: specify order number for limitated module usage
"<ORDER></ORDER>" ;<!--(optional for restricted customizations; missing statement makes module valid for all orders)-->
;
; Parameter Check <PARAn Name='aAbcdef' MIN='xxx' MAX='yyy' />  (watch for correct spacings and apostrophs!)
"<PARAMETER_CHK>"
"<PARA1 Name='iEng_Motortype' MIN='208' MAX='920' />"
"<PARA2 />"
"<PARA3 />"
"<PARA4 />"
"<PARA5 />"
"</PARAMETER_CHK>"
;
; Statement, that this module´s parameter check passing is mandatory (KN is allways mandatory, so other statements than TRUE here in this module are ignored)
"<MANDATORYMODULE>TRUE</MANDATORYMODULE>"
;
; Permanent Datamodule Filenames<!-- NAME ist ohne Dateiendung einzutragen; Nur für Counter und interne Parameter verwenden-->
"<DATAMODULES>" ;<!-- optional; mehrere DATAMODULES erlaubt-->
"	<DATAMODULE>par_KN</DATAMODULE>"
"</DATAMODULES>"
;
; Dependencies Modules (MMxx.yy.zz.cc)
"<DEPENDENCIES>"
"	<DEPENDENCY MODULE='SA' VERSION='04.14.00.00' />"
"	<DEPENDENCY MODULE='OP' VERSION='04.03.00.00' />"
"	<DEPENDENCY MODULE='AB' VERSION='04.03.00.00' />"
"	<DEPENDENCY MODULE='IG' VERSION='04.01.00.00' />"
"	<DEPENDENCY MODULE='KL' VERSION='04.03.00.00' />"
"	<DEPENDENCY MODULE='PB' VERSION='04.00.04.00' />"
"	<DEPENDENCY MODULE='VI' VERSION='04.00.00.00' />"
"	<DEPENDENCY MODULE='HA' VERSION='04.07.00.00' />"
"	<DEPENDENCY MODULE='EC' VERSION='04.14.00.00' />"
"	<DEPENDENCY MODULE='GT' VERSION='04.07.00.00' />"
"   <DEPENDENCY VISVERSION='02.15.00.00' />"			; Dependencies Visualization
"</DEPENDENCIES>"
;
; Module function description
"<MODULEFUNCTION>" ;<!-- short overview documentation of module function; add reference to detailed information, if available-->
"	<General>	"
"	Knocking Prevention "
"	</General>	"
""
"	<F1 Name='enter name of main function 1 here' LastModified='4.0.0.0'>"
"	o knocking monitoring with KLS90	"
"	</F1>"
"	<F3 Name='enter name of main function 2 here' LastModified='4.0.0.0'>"
"	o knocking monitoring with KLS98	"
"	</F2>"
"	<F3 Name='enter name of main function 3 here' LastModified='4.0.0.0'>"
"	o knocking monitoring with SAFIKLS	"
"	</F3>"
""
"	<Info>"
"	 V4.01.00.00	new interfaces added"
"	 V4.02.00.00	added safi dmr"
"	 V4.03.00.00	add MANDATORYMODULE statement"
"	 V4.04.00.00	versions changed"
" 	 V4.04.00.00	VISU knocking IP reduction"
"    V4.04.00.00    Bugfix: KLS98 validation - MSF not working "
"    V4.05.01.00    BU 01: change A3342 Knock sensor measuring sensor failure from Prio 3 to Prio 2"
" 	 V4.07.00.00	Added RKS package"
"	 V4.07.00.00	BU 01: avoiding division by 0"
"	<Customized LastModified='4.0.0.0'>	"
"	- Nothing "
"	</Customized>	"
""
"</MODULEFUNCTION>"
;
"</META>"
```

### module_Knocking.typ - Package data types
```iecst
(********************************************************************
 * COPYRIGHT -- INNIO Company
 ********************************************************************
 * Package: Knocking
 * File: module_Knocking.typ
 * Author: WaldharM
 * Created: October 03, 2011
 ********************************************************************
 * Data types of package Knocking
 ********************************************************************)

TYPE
	IN_KN_Struct : 	STRUCT  (* general*)
		tMS_PBC0 : ARRAY[0..12]OF _tSAFImdatas; (* Pressure based control measuring data 0*) (* OldName: DMR_md1; Cycle:2; *)
		tMS_PBC1 : ARRAY[0..12]OF _tSAFImdatas; (* Pressure based control measuring data 1 *) (* OldName: DMR_md1; Cycle:2; *)
		tMS_PBC2 : ARRAY[0..12]OF _tSAFImdatas; (* Pressure based control measuring data 2 *) (* OldName: DMR_md2; Cycle:2; *)
		tMS_PBC3 : ARRAY[0..12]OF _tSAFImdatas; (* Pressure based control measuring data 3 *) (* OldName: DMR_md3; Cycle:2; *)
		tMS_PBC4 : ARRAY[0..12]OF _tSAFImdatas; (* Pressure based control measuring data 4 *) (* OldName: DMR_md4; Cycle:2; *)
		tMS_PBC5 : ARRAY[0..12]OF _tSAFImdatas; (* Pressure based control measuring data 5 *) (* OldName: DMR_md5; Cycle:2; *)
		tMS_PBC6 : ARRAY[0..12]OF _tSAFImdatas; (* Pressure based control measuring data 6 *) (* OldName: DMR_md6; Cycle:2; *)
		tMS_PBC7 : ARRAY[0..12]OF _tSAFImdatas; (* Pressure based control measuring data 7 *) (* OldName: DMR_md7; Cycle:2; *)
		tMS_PBC8 : ARRAY[0..12]OF _tSAFImdatas; (* Pressure based control measuring data 8 *) (* OldName: DMR_md8; Cycle:2; *)
		tMS_PBC9 : ARRAY[0..12]OF _tSAFImdatas; (* Pressure based control measuring data 9 *) (* OldName: DMR_md9; Cycle:2; *)
		tMS_PBC10 : ARRAY[0..12]OF _tSAFImdatas; (* Pressure based control measuring data 10 *) (* OldName: DMR_md10; Cycle:2; *)
		tMS_PBC11 : ARRAY[0..12]OF _tSAFImdatas; (* Pressure based control measuring data 11 *) (* OldName: DMR_md11; Cycle:2; *)
		tMS_PBC12 : ARRAY[0..12]OF _tSAFImdatas; (* Pressure based control measuring data 12 *) (* OldName: DMR_md12; Cycle:2; *)
		tMS_PBC13 : ARRAY[0..12]OF _tSAFImdatas; (* Pressure based control measuring data 13 *) (* OldName: DMR_md13; Cycle:2; *)
		tMS_PBC14 : ARRAY[0..12]OF _tSAFImdatas; (* Pressure based control measuring data 14 *) (* OldName: DMR_md14; Cycle:2; *)
		tMS_PBC15 : ARRAY[0..12]OF _tSAFImdatas; (* Pressure based control measuring data 15 *) (* OldName: DMR_md15; Cycle:2; *)
		tMS_PBC16 : ARRAY[0..12]OF _tSAFImdatas; (* Pressure based control measuring data 16 *) (* OldName: DMR_md16; Cycle:2; *)
		tMS_PBC17 : ARRAY[0..12]OF _tSAFImdatas; (* Pressure based control measuring data 17 *) (* OldName: DMR_md17; Cycle:2; *)
		tMS_PBC18 : ARRAY[0..12]OF _tSAFImdatas; (* Pressure based control measuring data 18 *) (* OldName: DMR_md18; Cycle:2; *)
		tMS_PBC19 : ARRAY[0..12]OF _tSAFImdatas; (* Pressure based control measuring data 19 *) (* OldName: DMR_md19; Cycle:2; *)
		rP_Act_Norm_Filt : REAL; (* actual power related to rP_Nom filtered T=1s  [%/P_Nom] *) (* OldName: P_IST; Cycle:2; *)
		tAB2KN : AmmBase2MM; (* 0 *) (* OldName: 0; Cycle:2; *)
		rN_EngAct : REAL; (* engine speed *) (* OldName: n_ist; Cycle:2; *)
		iSt_OpMode : UDINT; (* engine operation mode *) (* OldName: 0; Cycle:2; *)
		tP_Act : ARRAY[0..2]OF HALioAi_Type; (* actual electric power [KW] *) (*OldName:ssPAct;Cycle:2;*)
		rP_Nom : REAL; (* nominal power *) (* OldName: 0; Cycle:2; *)
		rKLS98_X_Window1 : ARRAY[0..24]OF REAL; (* cylinder values of KLS98 window 1 *) (* OldName: Fenst1; Cycle:2; *)
		rKLS98_X_Window2 : ARRAY[0..24]OF REAL; (* cylinder values of KLS98 window 2 *) (* OldName: Fenst2; Cycle:2; *)
		rKLS98_X_Window3 : ARRAY[0..24]OF REAL; (* cylinder values of KLS98 window 3 *) (* OldName: Fenst3; Cycle:2; *)
		rKLS98_X_Window4 : ARRAY[0..24]OF REAL; (* cylinder values of KLS98 window 4 *) (* OldName: Fenst4; Cycle:2; *)
		tGCB_On_TC2 : HALioDi_Type; (* DI: Generator circuit breaker closed, TC2 synchron *) (* OldName: GCB_ON_TC1 ; Cycle:2; *)
		iU_SAFI_Win1 : ARRAY[0..24]OF INT; (* cylinder values of KLS window 1 *) (* OldName: Fenst1; Cycle:2; *)
		iU_SAFI_Win2 : ARRAY[0..24]OF INT; (* cylinder values of KLS window 2 *) (* OldName: Fenst2; Cycle:2; *)
		iU_SAFI_Win3 : ARRAY[0..24]OF INT; (* cylinder values of KLS window 3 *) (* OldName: Fenst3; Cycle:2; *)
		iU_SAFI_Win4 : ARRAY[0..24]OF INT; (* cylinder values of KLS window 4 *) (* OldName: Fenst4; Cycle:2; *)
		tPB2MM : ParaBase2MM_type; (* Messages from parametercheck module parameter are OK *) (* OldName: new PV; Cycle:2; *)
		tKLS90_1 : HALioAi_Type; (* AI: KLS90 sensor 1 signal *) (* OldName: ssKLS_Signal1; Cycle:2; *)
		tKLS90_2 : HALioAi_Type; (* AI: KLS90 sensor 1 signal *) (* OldName: ssKLS_Signal2; Cycle:2; *)
		tEng_Run : HALioDo_Type; (* engine operating state *) (* OldName: M_BTRB; Cycle:5; *)
		iIdx_OMSS : INT; (* index of operation mode selector switch *) (* OldName: BWS_HA; Cycle:2; *)
		iPassLevel : INT; (*pass level actual*) (*OldName:ucPassLevel; Cycle:5;*)
		bGasTyp1_Act : BOOL; (* gas type 1 active *) (*OldName:AN_GAS1,AW_ZZP1;Cycle:2;*)
		bGasTyp2_Act : BOOL; (* gas type 2 active *) (*OldName:AN_GAS2,AW_ZZP2;Cycle:2;*)
		bGasTyp3_Act : BOOL; (* gas type 3 active *) (*OldName:AN_GAS3,AW_ZZP3;Cycle:2;*)
		bGasTyp4_Act : BOOL; (* gas type 4 active *) (*OldName:AN_GAS4,AW_ZZP4;Cycle:2;*)
		bGasTypMix1_2_Act : BOOL; (* gas type mix 1-2 active *) (*OldName:AN_GAS1_2,AW_ZZP1_2;Cycle:2;*)
		bSCO_Active : BOOL; (* safety cut out gas valves glow ignition prevention *) (* OldName: SICH_SCHL; Cycle:5; *)
		bIPC_MSF : ARRAY[0..24]OF BOOL; (* in-cylinder pressure sensor measuring signal failure *) (* OldName: bDMRFault; Cycle: 2 *)
		bTimingRedActMx : ARRAY[0..24]OF BOOL; (* *) (* OldName: bTimingRedActMx; Cycle: 2 *)
		bKLS98_Fault : ARRAY[0..24]OF BOOL; (* TRUE= faulty cyl. knocking signal *) (*OldName:bKLS98Fault; Cycle: 2*)
		bKLS98_Signal : ARRAY[0..24]OF BOOL; (* KLS Measurement Signal Knock Sensor *) (*OldName:KLSMS; Cycle: 2*)
		bPBCSlowDriftCheck : ARRAY[0..24]OF BOOL; (* error info for PBC *) (* OldName: bPBCSlowDriftCheck; Cycle:2; *)
		iNum_KnckFiltEngCyc : INT; (* Engine cycles for knock containment V2*) (* OldName: newPV; Cycle: 2;*)
		rGT_RatioMix : REAL; (*Gas mixture rate after ramp fub [%], e.g. 0.5 = 50%*) (* OldName: 	ssRatioMix	; Cyclic:2; *)
		rGT_QualMix_1_2 : REAL; (*Mixture ratio bet. gas 1 and 2 [%], e.g. value 0.75 =75%*) (* OldName: 	ssMisch1_2	; Cyclic: ; *)
		bPBCSensErr : ARRAY[0..24]OF BOOL; (* error info for PBC *) (* OldName:bZM_PBCSensErr; Cycle:2 *)
		bPBCCompLineCheck : ARRAY[0..24]OF BOOL; (* error info for PBC *) (* OldName:bPBCCompLineCheck; Cycle:2 *)
		bPBCNegVoltCheck : ARRAY[0..24]OF BOOL; (* error info for PBC *) (* OldName:bPBCNegVoltCheck; Cycle:2 *)
		bPBCNegPresCheck : ARRAY[0..24]OF BOOL; (* error info for PBC *) (* OldName:bPBCNegPresCheck; Cycle:2 *)
		bPBCPresSlopeCheck : ARRAY[0..24]OF BOOL; (* error info for PBC *) (* OldName:bPBCPresSlopeCheck; Cycle:2 *)
		tiSFIKW_OffDelay : TIME; (* Hold On Delay for SFIKW Bit, default 100ms*) (* OldName: newPV; Cycle: 2;*)
		bPFPDR_Act : BOOL; (* PFPDR active *) (* OldName: new PV; Cycle: 2; *)
		bPFPDR_Knck_Slow : BOOL; (* PFPDR slow knock time *) (* OldName: new PV; Cycle: 2; *)
		bSimWinMOD_Active : BOOL; (*WinMOD simulation active*) (* OldName: new PV; Cycle: 5;*)
		PermRKS : tRKS_Perm; (* RKS Perm structure, values stored in EC Module *) (* OldName: newPV; Cycle: 2;*)
		bLimpHomeCylRKS : ARRAY[0..24]OF BOOL; (* Cylinders in LimpHomeRKS *) (* OldName: newPV; Cycle: 2;*)
		bSA_VCD_Active : BOOL; (*Enable visualization of VCD parameters for legacy versions*)
		bSA_Win1FrozenAltern : ARRAY[0..24]OF BOOL; (*Knock noise signal frozen or alternating*)
	END_STRUCT;
	tRKS_Perm : 	STRUCT
		bEna : BOOL; (* Enables RKS Knock Control *)
		iTable : ARRAY[0..15]OF USINT; (* Logic Table *)
		rCA_IP_Red : REAL;
		rDur_Downset : REAL; (* Duration downset in [%] *)
		iNum_EngCyc_Limp_Recover : INT; (* amount of engine cycles without limphom to switch to PBC *)
	END_STRUCT;
	OUT_KN_Struct : 	STRUCT  (* general*)
		tKN2AB : MM2AmmBase; (* 0 *) (* OldName: 0; Cycle:   *)
		iKls98_KnckValue_Max : UINT; (* maximum knocking value *) (* OldName: Fenst1Max ; Cycle: 2 *)
		iKls98_KnckValue_Min : UINT; (* minimum knocking value *) (* OldName: Fenst1Min ; Cycle: 2 *)
		iKls98_KnckValue_Avg : UINT; (* knocking value average *) (* OldName: Fenst1Avg ; Cycle: 2 *)
		iKls98_VNValue_Max : UINT; (* maximum valve noise *) (* OldName: Fenst2Max ; Cycle: 2 *)
		iKls98_VNValue_Min : UINT; (* minimum valve noise *) (* OldName: Fenst2Min ; Cycle: 2 *)
		iKls98_VNValue_Avg : UINT; (* valve noise average *) (* OldName: Fenst2Avg ; Cycle: 2 *)
		rKnck_Intgr_Max : REAL; (* maximum integrated knock value *) (* OldName: IntKlopfMx ; Cycle: 2 *)
		rKnck_Intgr_Min : REAL; (* minimum integrated knock value *) (* OldName: IntKlopfMn ; Cycle: 2 *)
		rKnck_Intgr_Avg : REAL; (* integrated knock value average  *) (* OldName: IntKlopfAv ; Cycle: 2 *)
		iIdx_Cyl_Knck_Max : INT; (* cyl. with highest knock signal *) (* OldName: ucKlopfMxZyl ; Cycle: 2 *)
		rKnck_Intgr : ARRAY[0..24]OF REAL; (* integrated cylinder knock values *) (* OldName: IntKlopf ; Cycle: 2 *)
		rKno_IP_Red : REAL; (* timing reduction by knocking *) (* OldName: klreg_dz ; Cycle: 2 *)
		rKno_P_Red : REAL; (* power red. by knocking *) (* OldName: klreg_dp ; Cycle: 2 *)
		rKno_T2s_Red : REAL; (* mixture temp. red. by knocking *) (* OldName: klreg_dt2 ; Cycle: 2 *)
		rP_Red_Knck_Norm : REAL; (* power reduction by knocking *) (* OldName: ssPowerRedKlopf ; Cycle: 2 *)
		rCA_Knck_Red : ARRAY[0..24]OF REAL; (* cylinder timing reduction by knocking *) (* OldName: ssKlRegdZZP ; Cycle: 2 *)
		bKLS98_MSF : ARRAY[0..24]OF BOOL; (* knocking sensor measuring signal failure *) (* OldName: bKLS98Fault; Cycle: 2 *)
		tKN2PB : MM2ParaBase_type; (* Data exchange structure to ParaBase *) (* OldName: new; Cycle: 5 *)
		rVNValue : ARRAY[0..24]OF REAL; (* cylinder values for valve noise *) (* OldName: Fenst2; Cycle: 2 *)
		rKnck_Noise : ARRAY[0..24]OF REAL; (* cylinder value for knocking noise *) (* OldName: Fenst1; Cycle: 2 *)
		rKnck_KPressure : ARRAY[0..24]OF REAL; (* cylinder value for knocking pressure *) (* OldName: Klopfen; Cycle: 2 *)
		tFastAO_KN_A : HALioAo_Type; (* fast analog output signals for validation *) (* OldName: AOFast_BuR_A; Cycle: 2 *)
		tFastAO_KN_B : HALioAo_Type; (* fast analog output signals for validation *) (* OldName: AOFast_BuR_B; Cycle: 2 *)
		rPr_Knck_Lim : ARRAY[0..24]OF REAL; (* knock limit*) (* OldName: knockFilt; Cycle 2;*)
		rPr_Knck_Filt : ARRAY[0..24]OF REAL; (* filtred knock signal with containment V2*) (* OldName: knockFilt; Cycle 2;*)
		iState_RKS : ARRAY[0..24]OF USINT; (* state for every cylinder, 1 = PBC, 2 = RKS, 3= FTC *) (* OldName: 0; Cycle:2; *)
		rPr_P2s_Knck_Offs : REAL; (* Offset for charge pressure due Knock *) (* OldName: 0; Cycle:2; *)
		rPmax_Knck_Red : ARRAY[0..24]OF REAL; (* cylinder Pmax reduction by knocking *) (* OldName: 0 ; Cycle: 2 *)
		rIntSignal : REAL; (*Knockintegrator level KLS90*)
		bTExh_Mon_UseNarrowWindow : ARRAY[0..24]OF BOOL; (*narrower threshold activation for exhaust temperature monitoring*)
		bP_Red_SAErr : BOOL; (*Trigger SAFI power reduction*)
		bKnockSig : ARRAY[0..24]OF BOOL; (*SAFI KLS measurement signal error [-]*)
	END_STRUCT;
	Para_Struct : 	STRUCT
		rKno_IP_Red_StP : REAL; (* start point for ignition point reduction for knocking   *) (* OldName: kl_dz_li ; Cycle:   *)
		rKno_IP_Red_EnP : REAL; (*  end point for ignition point reduction for knocking   *) (* OldName: kl_dz_e ; Cycle:   *)
		rKno_P_Red_StP : REAL; (*  start point power reduction for knocking   *) (* OldName: kl_dp_li ; Cycle:   *)
		rKno_P_Red_EnP : REAL; (*  end point power reduction for knocking   *) (* OldName: kl_dp_e ; Cycle:   *)
		rKno_T2s_Red_StP : REAL; (*  start point t2s reduction for knocking   *) (* OldName: kl_dt2_li ; Cycle:   *)
		rKno_T2s_Red_EnP : REAL; (*  end point t2s reduction for knocking   *) (* OldName: kl_dt2_e ; Cycle:   *)
		bKLS98_Active : BOOL; (*  TRUE = KLS98 active  *) (* OldName: kls98_vis ; Cycle:   *)
		tiKnck_Intgr_Down : TIME; (*PARA [12084]: knock integrator decreasing factor  *) (* OldName: int_down ; Cycle:   *)
		tiKnck_Intgr_Up : TIME; (*PARA [12085]: knock integrator increasing factor  *) (* OldName: int_up; Cycle:   *)
		tiKnck_Intgr_Up_CylOpt : TIME; (*PARA [12086]: knock integrator increasing factor for timing point optimisation  *) (* OldName: int_up_CylOpt ; Cycle:   *)
		iKlS_KnckValue_Limit : UINT; (*  limit for knocking detection [mV]  *) (* OldName: Fenst2LiMx ; Cycle:   *)
		rCA_Ign_OP_Max : ARRAY[0..4]OF REAL; (*  maximum allowed ingnition point  *) (* OldName: ssMinKlZZP ; Cycle:   *)
		rU_Knck_Lim : REAL; (*  limit value for knock detection  *) (* OldName: KlopfLimit ; Cycle:   *)
		rP_Eng_KC_Act_Lim : REAL; (* power output start knock control *) (* OldName: klopf_akt ; Cycle:   *)
		rP_Knck_Act_Hy : REAL; (*  hyst power start knock control   *) (* OldName: klopf_hys ; Cycle:   *)
		bIgnP_Opt_Exist : BOOL; (*  TURE =  igniton timing point optimisation is active  *) (* OldName: bCylOpt ; Cycle:   *)
		bSA_PBC_Active : BOOL; (*PARA [12119]: TRUE = SAFI PBC function is enabled/active  *) (* OldName: bSAFIDMR_Act; Cycle:   *)
		bSA_KLS_Active : BOOL; (*PARA [12118]: TRUE = SAFI KLS function is enabled/active *) (* OldName: bSAFIKLS_Act; Cycle: 0 *)
		bKLS90_Exist : BOOL; (* Para: TRUE = KLS90 is enabled/active  *) (* OldName: 0; Cycle: 0 *)
		iKlS_MSFailure_Limit : UINT; (*PARA [12074]: limit for measuring signal failue [mV]  *) (* OldName: Fenst2LiMn; Cycle: 0 *)
		rKLS90_KnckValue_LimitB : REAL; (*PARA [14505]: limit for KLS90 knocking detection - BankB [mA] *) (* OldName: kl_limit_1, kl_limit_2; Cycle: 0 *)
		rKLS90_KnckValue_Limit : REAL; (*PARA [12075]: limit for KLS90 knocking detection - BankA [mA] *) (* OldName: kl_limit_1, kl_limit_2; Cycle: 0 *)
		iEng_Motortype : INT; (* 0 *) (* OldName: 0; Cycle: 0 *)
		bGlowIgnPrevActive : BOOL; (*PARA [12089]: TRUE = glow ignition prevention activ *) (* OldName: sel_GlowIgnPrevent; Cycle: 2 *)
		rPr_PBC_Knck_Lim : REAL; (*PARA [12776]: PBC Knock Limit [bar] *) (* OldName: KlopfLimitDMR; Cycle: 2 *)
		rN_EngNom : REAL; (* nominal speed *) (* OldName: n_nenn ; Cycle: 2 *)
		bSA_PI_Active : BOOL; (*PARA [12120]: TRUE = SAFI port injection is enabled/active  *) (* OldName: bSAFIPI_Act; Cycle: 2 *)
		rKno_Int_MinLim : REAL; (*PARA [13460]: lower knock integrator limit for PI Engines *)
		rKno_IP_Scale_StP : REAL; (*PARA [13461]: start point for ignition timing point scaling for knocking   *)
		rCA_IP_Knck_Max : REAL; (*PARA [13466]: maximum ignition timing point reduction *)
		rKno_Pmax_Red_StP : REAL; (*PARA [13462]: start point for Pmax reduction for knocking   *) (* OldName: newPV ; Cycle:   *)
		rKno_Pmax_Red_EnP_dlt : REAL; (*PARA [13463]: end point for Pmax reduction for knocking   *) (* OldName: newPV ; Cycle:   *)
		rPmax_Knck_Max : REAL; (*PARA [13468]: maximum Pmax reduction *)
		rKno_P2s_Inc_StP : REAL; (*PARA [13464]: start point for charging pressure increase for knocking   *) (* OldName: newPV ; Cycle:   *)
		rKno_P2s_Inc_EnP : REAL; (*PARA [13465]: end point for charging pressure increase for knocking   *) (* OldName: newPV ; Cycle:   *)
		rPr_P2s_Knck_Max : REAL; (*PARA [13467]: maximum charging pressure increase *)
		iKno_Pmax_CylMax : USINT; (*PARA [13469]: max number of cylinders for Pmax reduction *)
		rPr_PBC_Knck_Heavy : REAL; (*PARA [13501]: PBC Heavy Knock Limit [bar] *) (* OldName: newPV; Cycle: 2 *)
		bType6BlockAfterTrip : BOOL; (*BOOL: Block Engine after Knock trip in combination with measurung signal failure knock sensor (type 6 only)*)
		bMeNoi_Activation : BOOL; (*Para [14415]: Mechanical noise monitoring active*)
		rP_Marg_MeNoiAL_Dev : REAL; (*Para [14417]: Deviation limit to apply increased temperature monitoring sensitivity*)
		rFiltTimeCnt_MeNoi : REAL; (*Para [14416]: Filter constant operation point detection*)
		bSA_Ign_Active : BOOL; (*PARA [12117]: TRUE = SAFI ignition function is enabled/active  *)
	END_STRUCT;
	MM2VIS_Struct : 	STRUCT  (*OPC variables from module to VIS*)
		bMeNoi_Mon_vis : BOOL; (*Activation MeNoi Mon Para folder in HMI*)
		bMsg3053 : BOOL; (* Trip: KLS valve noise cylinder 1 *) (* OldName: KLSVEN[1]; Cycle: 0 *)
		bMsg3054 : BOOL; (* Trip: KLS valve noise cylinder 2 *) (* OldName: KLSVEN[2]; Cycle: 0 *)
		bMsg3055 : BOOL; (* Trip: KLS valve noise cylinder 3 *) (* OldName: KLSVEN[3]; Cycle: 0 *)
		bMsg3056 : BOOL; (* Trip: KLS valve noise cylinder 4 *) (* OldName: KLSVEN[4]; Cycle: 0 *)
		bMsg3057 : BOOL; (* Trip: KLS valve noise cylinder 5 *) (* OldName: KLSVEN[5]; Cycle: 0 *)
		bMsg3058 : BOOL; (* Trip: KLS valve noise cylinder 6 *) (* OldName: KLSVEN[6]; Cycle: 0 *)
		bMsg3059 : BOOL; (* Trip: KLS valve noise cylinder 7 *) (* OldName: KLSVEN[7]; Cycle: 0 *)
		bMsg3060 : BOOL; (* Trip: KLS valve noise cylinder 8 *) (* OldName: KLSVEN[8]; Cycle: 0 *)
		bMsg3061 : BOOL; (* Trip: KLS valve noise cylinder 9 *) (* OldName: KLSVEN[9]; Cycle: 0 *)
		bMsg3062 : BOOL; (* Trip: KLS valve noise cylinder 10 *) (* OldName: KLSVEN[10]; Cycle: 0 *)
		bMsg3063 : BOOL; (* Trip: KLS valve noise cylinder 11 *) (* OldName: KLSVEN[11]; Cycle: 0 *)
		bMsg3064 : BOOL; (* Trip: KLS valve noise cylinder 12 *) (* OldName: KLSVEN[12]; Cycle: 0 *)
		bMsg3065 : BOOL; (* Trip: KLS valve noise cylinder 13 *) (* OldName: KLSVEN[13]; Cycle: 0 *)
		bMsg3066 : BOOL; (* Trip: KLS valve noise cylinder 14 *) (* OldName: KLSVEN[14]; Cycle: 0 *)
		bMsg3067 : BOOL; (* Trip: KLS valve noise cylinder 15 *) (* OldName: KLSVEN[15]; Cycle: 0 *)
		bMsg3068 : BOOL; (* Trip: KLS valve noise cylinder 16 *) (* OldName: KLSVEN[16]; Cycle: 0 *)
		bMsg3069 : BOOL; (* Trip: KLS valve noise cylinder 17 *) (* OldName: KLSVEN[17]; Cycle: 0 *)
		bMsg3070 : BOOL; (* Trip: KLS valve noise cylinder 18 *) (* OldName: KLSVEN[18]; Cycle: 0 *)
		bMsg3071 : BOOL; (* Trip: KLS valve noise cylinder 19 *) (* OldName: KLSVEN[19]; Cycle: 0 *)
		bMsg3072 : BOOL; (* Trip: KLS valve noise cylinder 20 *) (* OldName: KLSVEN[20]; Cycle: 0 *)
		bMsg3073 : BOOL; (* Trip: KLS98 knocking failure cylinder 1 *) (* OldName: KLOPF[1]; Cycle: 0 *)
		bMsg3074 : BOOL; (* Trip: KLS98 knocking failure cylinder 2 *) (* OldName: KLOPF[2]; Cycle: 0 *)
		bMsg3075 : BOOL; (* Trip: KLS98 knocking failure cylinder 3 *) (* OldName: KLOPF[3]; Cycle: 0 *)
		bMsg3076 : BOOL; (* Trip: KLS98 knocking failure cylinder 4 *) (* OldName: KLOPF[4]; Cycle: 0 *)
		bMsg3077 : BOOL; (* Trip: KLS98 knocking failure cylinder 5 *) (* OldName: KLOPF[5]; Cycle: 0 *)
		bMsg3078 : BOOL; (* Trip: KLS98 knocking failure cylinder 6 *) (* OldName: KLOPF[6]; Cycle: 0 *)
		bMsg3079 : BOOL; (* Trip: KLS98 knocking failure cylinder 7 *) (* OldName: KLOPF[7]; Cycle: 0 *)
		bMsg3080 : BOOL; (* Trip: KLS98 knocking failure cylinder 8 *) (* OldName: KLOPF[8]; Cycle: 0 *)
		bMsg3081 : BOOL; (* Trip: KLS98 knocking failure cylinder 9 *) (* OldName: KLOPF[9]; Cycle: 0 *)
		bMsg3082 : BOOL; (* Trip: KLS98 knocking failure cylinder 10 *) (* OldName: KLOPF[10]; Cycle: 0 *)
		bMsg3083 : BOOL; (* Trip: KLS98 knocking failure cylinder 11 *) (* OldName: KLOPF[11]; Cycle: 0 *)
		bMsg3084 : BOOL; (* Trip: KLS98 knocking failure cylinder 12 *) (* OldName: KLOPF[12]; Cycle: 0 *)
		bMsg3085 : BOOL; (* Trip: KLS98 knocking failure cylinder 13 *) (* OldName: KLOPF[13]; Cycle: 0 *)
		bMsg3086 : BOOL; (* Trip: KLS98 knocking failure cylinder 14 *) (* OldName: KLOPF[14]; Cycle: 0 *)
		bMsg3087 : BOOL; (* Trip: KLS98 knocking failure cylinder 15 *) (* OldName: KLOPF[15]; Cycle: 0 *)
		bMsg3088 : BOOL; (* Trip: KLS98 knocking failure cylinder 16 *) (* OldName: KLOPF[16]; Cycle: 0 *)
		bMsg3089 : BOOL; (* Trip: KLS98 knocking failure cylinder 17 *) (* OldName: KLOPF[17]; Cycle: 0 *)
		bMsg3090 : BOOL; (* Trip: KLS98 knocking failure cylinder 18 *) (* OldName: KLOPF[18]; Cycle: 0 *)
		bMsg3091 : BOOL; (* Trip: KLS98 knocking failure cylinder 19 *) (* OldName: KLOPF[19]; Cycle: 0 *)
		bMsg3092 : BOOL; (* Trip: KLS98 knocking failure cylinder 20 *) (* OldName: KLOPF[20]; Cycle: 0 *)
		bMsg3279 : BOOL; (* OP Message: Knocking failure *) (* OldName: bBKnockErr; Cycle: 0 *)
		bMsg3281 : BOOL; (* OP Message: Valve noise high *) (* OldName: bBValveErr; Cycle: 0 *)
		bMsg3282 : BOOL; (* OP Message: Knock sensor measuring signal failure *) (* OldName: bBKnockSigErr; Cycle: 0 *)
		bMsg3339 : BOOL; (* Trip: Knocking failure *) (* OldName: bAKnockErr; Cycle: 0 *)
		bMsg3341 : BOOL; (* Trip: Valve noise high *) (* OldName: bAKnockErr; Cycle: 0 *)
		bMsg3342 : BOOL; (* Trip: Knock sensor measuring sensor failure *) (* OldName: bAKnockSigErr; Cycle: 0 *)
		bMsg3541 : BOOL; (* Warning: Knock sensor measuring sensor failure *) (* OldName: bWKnockSigErr; Cycle: 0 *)
		iKls98_KnckValue_Max : UINT; (* maximum knocking value *) (* OldName: Fenst1Max ; Cycle: 0 *)
		iKls98_KnckValue_Min : UINT; (* minimum knocking value *) (* OldName: Fenst1Min ; Cycle: 0 *)
		iKls98_KnckValue_Avg : UINT; (* knocking value average *) (* OldName: Fenst1Avg ; Cycle: 0 *)
		iKls98_VNValue_Max : UINT; (* maximum valve noise *) (* OldName: Fenst2Max ; Cycle: 0 *)
		iKls98_VNValue_Min : UINT; (* minimum valve noise *) (* OldName: Fenst2Min ; Cycle: 0 *)
		iKls98_VNValue_Avg : UINT; (* valve noise average *) (* OldName: Fenst2Avg ; Cycle: 0 *)
		rKnck_Intgr_Max : REAL; (* maximum integrated knock value *) (* OldName: IntKlopfMx ; Cycle: 0 *)
		rKnck_Intgr_Min : REAL; (* minimum integrated knock value *) (* OldName: IntKlopfMn ; Cycle: 0 *)
		rKnck_Intgr_Avg : REAL; (* integrated knock value average  *) (* OldName: IntKlopfAv ; Cycle: 0 *)
		iIdx_Cyl_Knck_Max : INT; (* cyl. with highest knock signal *) (* OldName: ucKlopfMxZyl ; Cycle: 0 *)
		rKnck_Intgr : ARRAY[0..24]OF REAL; (* integrated cylinder knock values *) (* OldName: IntKlopf ; Cycle: 0 *)
		rKno_IP_Red : REAL; (* timing reduction by knock permill *) (* OldName: klreg_dz ; Cycle: 0 *)
		rKno_P_Red : REAL; (* power red. by knocking *) (* OldName: klreg_dp ; Cycle: 0 *)
		rKno_T2s_Red : REAL; (* mixture temp. red. by knocking *) (* OldName: klreg_dt2 ; Cycle: 0 *)
		rP_Red_Knck_Norm : REAL; (* power reduction by knocking *) (* OldName: ssPowerRedKlopf ; Cycle: 0 *)
		rCA_Knck_Red : ARRAY[0..24]OF REAL; (* cylinder timing reduction *) (* OldName: ssKlRegdZZP ; Cycle: 0 *)
		iMsg3279 : INT; (* ACM: Knocking failure *) (* OldName: iIdx_Err_Knock; Cycle: 0 *)
		iMsg3281 : INT; (* ACM: Vavle noise high *) (* OldName: iIdx_Err_Valve; Cycle: 0 *)
		iMsg3282 : INT; (* ACM: Knock sensor measuring signal failure *) (* OldName: iIdx_Err_KnockSig; Cycle: 0 *)
		rVNValue : ARRAY[0..24]OF REAL; (* cylinder values for valve noise *) (* OldName: Fenst2; Cycle: 0 *)
		rKnck_Noise : ARRAY[0..24]OF REAL; (* cylinder value for knocking noise *) (* OldName: Fenst1; Cycle: 0 *)
		rKnck_KPressure : ARRAY[0..24]OF REAL; (* cylinder value for knocking noise *) (* OldName: Klopfen; Cycle: 0 *)
		rKLS90_Knck_Noise_1 : REAL; (* KLS90 cylinder 1 value for knocking noise  *) (* OldName: kl_ist_1; Cycle: 0 *)
		rKLS90_Knck_Noise_2 : REAL; (* KLS90 cylinder 2 value for knocking noise  *) (* OldName: kl_ist_2; Cycle: 0 *)
		bMsg1081 : BOOL; (* Trip: Knock sensor measuring signal failure KLS90 *) (* OldName: new PV; Cycle: 0 *)
		bMsg2111 : BOOL; (* Warning: Knock sensor measuring signal failure KLS90 *) (* OldName: new PV; Cycle: 0 *)
		bMsg1048 : BOOL; (* Trip: Knocking failure KLS90 *) (* OldName: new PV; Cycle: 0 *)
		rKnck_Noise_Avg : REAL; (* average value for knocking noise *) (* OldName: Fenst1Avg; Cycle: 0 *)
		rKnck_Noise_Max : REAL; (* maximum value for knocking noise *) (* OldName: Fenst1Max; Cycle: 0 *)
		rKnck_Noise_Min : REAL; (* minimum value for knocking noise *) (* OldName: Fenst1Min; Cycle: 0 *)
		bMsg2492 : BOOL; (*W2492 - Knocking in combination with a knock sensor failure – contact the service hotline*)
		iRKS_KnckSens_Color : ARRAY[0..24]OF INT;
		bMsg2440 : BOOL; (* W2440: RKS G2 unit Bank A CAN signal failure *) (* OldName: new PV; Cycle: 0 *)
		bMsg2441 : BOOL; (* W2441: RKS G2 unit Bank B CAN signal failure *) (* OldName: new PV; Cycle: 0 *)
		bKLS90_2_Exist: BOOL; (* Enables 2nd KLS90 sensor on HMI *)
	END_STRUCT;
	_tSAFImdatas : 	STRUCT
		data1 : UINT;
		data2 : UINT;
		data3 : UINT;
	END_STRUCT;
	_tSAFIHardware : 	STRUCT
		HW_OPTION : USINT;
		HW_VERSION : USINT;
	END_STRUCT;
	tPIopen : 	STRUCT
		timing : UINT;
		duration : UINT;
	END_STRUCT;
	rtctime_typ : 	STRUCT
		year : UINT;
		month : USINT;
		day : USINT;
		reserve : USINT;
		hour : USINT;
		minute : USINT;
		second : USINT;
		millisec : UINT;
		microsec : UINT;
	END_STRUCT;
END_TYPE
```

### module_Knocking.var - Package variables
```iecst
(********************************************************************
 * COPYRIGHT -- INNIO Company
 ********************************************************************
 * Package: Knocking
 * File: module_Knocking.var
 * Author: WaldharM
 * Created: October 03, 2011
 ********************************************************************
 * Variables of package Knocking
 ********************************************************************)
VAR
	usFreig_n : UINT;
	ucKlopfMxZyl : USINT;
	ssMinKlZZP : ARRAY[0..4] OF INT;
	ssKlRegdZZP : ARRAY[0..25] OF INT;
	PN_GASART : INT;
	Para : Para_Struct;
	ParaFactoryDefault : Para_Struct := (0); (*First Init Values*)
	pm : Para_Struct;
	p_ist : INT;
	OUT_KN : OUT_KN_Struct;
	KLSVEN : ARRAY[0..25] OF BOOL;
	klreg_dz : INT;
	klreg_dt2 : INT;
	klreg_dp : INT;
	Klopflimit : INT;
	klopf_akt : INT;
	KLOPF : ARRAY[0..24] OF BOOL;
	kl_dz_li : INT;
	kl_dz_k : INT;
	kl_dz_e : INT;
	kl_dt2_li : INT;
	kl_dt2_k : INT;
	kl_dt2_e : INT;
	kl_dp_li : INT;
	kl_dp_k : INT;
	kl_dp_e : INT;
	IntKlopfMx : INT;
	IntKlopfMn : INT;
	IntKlopf : ARRAY[0..25] OF INT;
	IN_KN : IN_KN_Struct;
	iIdx_Err_Valve : USINT;
	iIdx_Err_KnockSig : USINT;
	iIdx_Err_Knock : USINT;
	Fenst4 : ARRAY[0..24] OF UINT; (*cylinder values of KLS98 window 4*)
	Fenst3 : ARRAY[0..24] OF UINT; (*cylinder values of KLS98 window 3*)
	Fenst2Min : UINT;
	Fenst2Max : UINT;
	Fenst2LiMx : UINT;
	Fenst2Avg : UINT;
	Fenst2 : ARRAY[0..24] OF UINT; (*cylinder values of KLS98 window 2*)
	Fenst1Min : UINT;
	Fenst1Max : UINT;
	Fenst1Avg : UINT;
	Fenst1 : ARRAY[0..24] OF UINT; (*cylinder values of KLS98 window 1*)
	bWKnockSigErr : BOOL;
	bMsg3541 : BOOL; (* Warning: Knock sensor measuring sensor failure *)
	bMsg3341 : BOOL; (* Trip: Valve noise high *)
	bMsg3339 : BOOL; (* Trip: Knocking failure *)
	bMsg3282 : BOOL; (* OP Message: Knock sensor measuring signal failure *)
	bMsg3281 : BOOL; (* OP Message: Valve noise high *)
	bMsg3279 : BOOL; (* OP Message: Knocking failure *)
	bMsg3092 : BOOL; (* Trip: KLS98 knocking failure cylinder 20 *)
	bMsg3091 : BOOL; (* Trip: KLS98 knocking failure cylinder 19 *)
	bMsg3090 : BOOL; (* Trip: KLS98 knocking failure cylinder 18 *)
	bMsg3089 : BOOL; (* Trip: KLS98 knocking failure cylinder 17 *)
	bMsg3088 : BOOL; (* Trip: KLS98 knocking failure cylinder 16 *)
	bMsg3087 : BOOL; (* Trip: KLS98 knocking failure cylinder 15 *)
	bMsg3086 : BOOL; (* Trip: KLS98 knocking failure cylinder 14 *)
	bMsg3085 : BOOL; (* Trip: KLS98 knocking failure cylinder 13 *)
	bMsg3084 : BOOL; (* Trip: KLS98 knocking failure cylinder 12 *)
	bMsg3083 : BOOL; (* Trip: KLS98 knocking failure cylinder 11 *)
	bMsg3082 : BOOL; (* Trip: KLS98 knocking failure cylinder 10 *)
	bMsg3081 : BOOL; (* Trip: KLS98 knocking failure cylinder 9 *)
	bMsg3080 : BOOL; (* Trip: KLS98 knocking failure cylinder 8 *)
	bMsg3079 : BOOL; (* Trip: KLS98 knocking failure cylinder 7 *)
	bMsg3078 : BOOL; (* Trip: KLS98 knocking failure cylinder 6 *)
	bMsg3077 : BOOL; (* Trip: KLS98 knocking failure cylinder 5 *)
	bMsg3076 : BOOL; (* Trip: KLS98 knocking failure cylinder 4 *)
	bMsg3075 : BOOL; (* Trip: KLS98 knocking failure cylinder 3 *)
	bMsg3074 : BOOL; (* Trip: KLS98 knocking failure cylinder 2 *)
	bMsg3073 : BOOL; (* Trip: KLS98 knocking failure cylinder 1 *)
	bMsg3072 : BOOL; (* Trip: KLS valve noise cylinder 20 *)
	bMsg3071 : BOOL; (* Trip: KLS valve noise cylinder 19 *)
	bMsg3070 : BOOL; (* Trip: KLS valve noise cylinder 18 *)
	bMsg3069 : BOOL; (* Trip: KLS valve noise cylinder 17 *)
	bMsg3068 : BOOL; (* Trip: KLS valve noise cylinder 16 *)
	bMsg3067 : BOOL; (* Trip: KLS valve noise cylinder 15 *)
	bMsg3066 : BOOL; (* Trip: KLS valve noise cylinder 14 *)
	bMsg3065 : BOOL; (* Trip: KLS valve noise cylinder 13 *)
	bMsg3064 : BOOL; (* Trip: KLS valve noise cylinder 12 *)
	bMsg3063 : BOOL; (* Trip: KLS valve noise cylinder 11 *)
	bMsg3062 : BOOL; (* Trip: KLS valve noise cylinder 10 *)
	bMsg3061 : BOOL; (* Trip: KLS valve noise cylinder 9 *)
	bMsg3060 : BOOL; (* Trip: KLS valve noise cylinder 8 *)
	bMsg3059 : BOOL; (* Trip: KLS valve noise cylinder 7 *)
	bMsg3058 : BOOL; (* Trip: KLS valve noise cylinder 6 *)
	bMsg3057 : BOOL; (* Trip: KLS valve noise cylinder 5 *)
	bMsg3056 : BOOL; (* Trip: KLS valve noise cylinder 4 *)
	bMsg3055 : BOOL; (* Trip: KLS valve noise cylinder 3 *)
	bMsg3054 : BOOL; (* Trip: KLS valve noise cylinder 2 *)
	bMsg3053 : BOOL; (* Trip: KLS valve noise cylinder 1 *)
	bKlopfregAkt : BOOL;
	bGnlWarning_modlKN : BOOL;
	bGnlTrip3_modlKN : BOOL;
	bGnlTrip2_modlKN : BOOL;
	bGnlTrip1_modlKN : BOOL;
	bBValveErr : BOOL;
	bBKnockSigErr : BOOL;
	bBKnockErr : BOOL;
	bAValveErr : BOOL;
	bAKnockSigErr : BOOL;
	bAKnockErr : BOOL;
	ssKLS_Signal1 : INT;
	ssKLS_Signal2 : INT;
	bKLS_Signal2_OK : BOOL; (*KN Sens 2 - Quality Signal*)
	int_down : INT;
	int_up : INT;
	RPSW6 : BOOL;
	Fenst2LiMn : UINT;
	MM2VIS : MM2VIS_Struct;
	xEngType : EngType;
	iMsg3279 : INT; (* ACM: Knocking failure *)
	iMsg3281 : INT; (* ACM: Vavle noise high *)
	iMsg3282 : INT; (* ACM: Knock sensor measuring signal failure *)
	bNoInitDetected : BOOL := FALSE; (*allways true, except 1cycle on init up*)
	bMsg1081 : BOOL;
	bMsg2111 : BOOL;
	RPSW_6 : BOOL;
	AN_KLOPF : BOOL;
	bMsg1048 : BOOL;
	RPSA_8 : BOOL;
	IntKlopfAv : INT;
	bMsg3342 : BOOL;
	bADMRSErr : BOOL; (* Trip: A3339 Knocking failure *)
	bMsg3339_Reset : BOOL := FALSE;
	KlopfLimitDMR : UINT; (* Para *)
	bBDMRSErr : BOOL;
	bKLSAFIFault : ARRAY[0..24] OF BOOL; (*oldname: bKLS98Fault*)
	ucZZPArt : USINT;
	tRealTime : rtctime_typ;
	xMeNoiAL : fMeNoiAL := (0); (*FuB*)
	bKnockSig : ARRAY[0..24] OF BOOL;
	rInt_Knck : ARRAY[0..24] OF REAL; (* knock integrator for PBC *)
	iState_RKS_old : ARRAY[0 .. 24] OF USINT; (* old state of RKS for every cylinder, 1 = PBC, 2 = RKS, 3= FTC*)
END_VAR
```

### Program Logical/Knocking/IN_Knck (IEC) - + IN task of knocking modul

- IN_KnckCyclic.st (not readable text: treated as protected, skipped)

#### IN_Knck.var - Local variables
```iecst
(********************************************************************
 * COPYRIGHT -- INNIO Company
 ********************************************************************
 * Program: IN_Knck
 * File: IN_Knck.var
 * Author: WaldharM
 * Created: October 03, 2011
 ********************************************************************
 * Local variables of program IN_Knck
 ********************************************************************)
VAR
	ucCylinderCount : USINT;
	ucGasTypCount : USINT;
	rCA_Ign_OP_Max_0 : REAL;
	DTGetTime_RPS : DTGetTime;
END_VAR
```

### Program Logical/Knocking/Kn_knock (IEC) - + knock monitoring with KLS90

- Kn_knockCyclic.st (not readable text: treated as protected, skipped)

- Kn_knockInit.st (not readable text: treated as protected, skipped)

#### Kn_knock.var
```iecst
VAR
	ssKLS1_Old : INT; (* signal last duration KLS90 sensor1 *)
	ssKLS2_Old : INT; (* signal last duration KLS90 sensor2 *)
	ssKLS_Signal : INT; (* scaled signal KLS90 sensor max *)
	ssIntSignal : INT; (* knocking integration signal *)
	fIntSignal : REAL; (* integrator of the KLS90 signal *)
	bSensor1OK : BOOL; (* signal KLS90 sensor 1 is ok *)
	bSensor2OK : BOOL; (* signal KLS90 sensor 2 is ok *)
	bKlopf1 : BOOL; (* knocking detection KLS90 sensor 1 *)
	bKlopf2 : BOOL; (* knocking detection KLS90 sensor 2 *)
	FILTER_KLS2 : FILTER; (* LP-filter signal KLS90 sensor 2 *)
	FILTER_KLS1 : FILTER; (* LP-filter signal KLS90 sensor 1 *)
	TP_KnockLow : TP; (* timer for low knock sensitivity *)
	TON_GETsignal : TON; (* time delay for GET signal failure *)
	ssMinIntKlopf : INT;
	ssMinIntKl : INT;
	TON_Nocksignal : TON; (* knock signal failure after 24h *)
	xOpMode : OpMode;
END_VAR
```

### Program Logical/Knocking/Knck_KLS98 (IEC) - + knock monitoring with KLS98

- Knck_KLS98Cyclic.st (not readable text: treated as protected, skipped)

- Knck_KLS98Init.st (not readable text: treated as protected, skipped)

#### Knck_KLS98.var - Local variables
```iecst
(********************************************************************
 * COPYRIGHT -- INNIO Company
 ********************************************************************
 * Program: Knck_KLS_98
 * File: Knck_KLS_98.var
 * Author: WaldharM
 * Created: October 03, 2011
 ********************************************************************
 * Local variables of program Knck_KLS_98
 ********************************************************************)
VAR
	KLimitVar : ARRAY[0..24] OF UINT; (* individual knock limit *)
	lIntKlopfAvg : DINT; (* sample average knock signal *)
	slFenst2LiMx : DINT; (* limit for knock detection [mV] *)
	ssMinIntKl : INT; (* temporary memory *)
	ssMinIntKlopf : INT; (* minimum allowed knock integrator *)
	ssRestIntDown : ARRAY[0..24] OF UINT; (* remainder of knock integrators *)
	ssRestIntUp : ARRAY[0..24] OF UINT; (* remainder of knock integrators *)
	TON_DecPowerRed : TON; (* FUB timer decrement misfire power *)
	TP_LowKnockLimit : TP; (* FUB timer for low knock limit *)
	ucCylinderCount : USINT; (* loop counter for cylinder number *)
	ucFenst2Cnt : USINT; (* sample counter valve noise values *)
	ucFenst2LimitCount : ARRAY[0..24] OF USINT;
	ucKlopfSensorCount : USINT; (* counter actual active knock sensor *)
	ulFenst1Avg : UDINT; (* sample average of knock noise *)
	ulFenst2Avg : UDINT; (* sample average of valve noise *)
	rFilt_Fenst1 : ARRAY[0..24] OF REAL; (* used for individual knock limit *)
	rGainFactor : REAL; (* individual knock limit gain factor *)
	rFilterFactor : REAL; (* time constant knock signal filter *)
	usFenst1 : UINT;
	usKLmin : UINT;
	rOff : REAL; (* individual knock limit offset *)
	xOpMode : OpMode; (*	bKlopfregAkt : BOOL;*) (*	klopf_hys : INT;*)
END_VAR
```

### Program Logical/Knocking/Kn_safi_kls (IEC) - + knock monitoring with SAFI-KLS

- Kn_safi_klsCyclic.st (not readable text: treated as protected, skipped)

- Kn_safi_klsInit.st (not readable text: treated as protected, skipped)

#### Kn_safi_kls.var - Local variables
```iecst
(********************************************************************
 * COPYRIGHT -- INNIO Company
 ********************************************************************
 * Program: Knck_safi_kls
 * File: Knck_safi_kls.var
 * Author: WaldharM
 * Created: October 10, 2011
 ********************************************************************
 * Local variables of program Knck_safi_kls
 ********************************************************************)
VAR
	ZMInKlopf : INT;
	usKLmin : UINT;
	usFenst1 : UINT;
	ulFenst2Avg : UDINT;
	ulFenst1Avg : UDINT;
	ucNrOfFaultKLSAFI : USINT;
	ucKLSMScount : ARRAY[0..24] OF USINT;
	ucKlopfSensorCount : USINT;
	ucFenst2LimitCount : ARRAY[0..24] OF USINT;
	ucFenst2Cnt : USINT;
	ucCylinderCount : USINT;
	TP_LowKnockLimit : TP;
	TON_SecondTick : TON;
	xTON_OffsKl : TON;
	ssRestIntUp : ARRAY[0..24] OF DINT;
	ssRestIntDown : ARRAY[0..24] OF DINT;
	ssMinIntKlopf : INT;
	ssMinIntKl : INT;
	slFenst2LiMx : DINT;
	lIntKlopfAvg : DINT;
	KLimitVar : ARRAY[0..24] OF UINT;
	IntKlopfMxOff : INT;
	bValve : ARRAY[0..24] OF BOOL;
	bReleaseOffsKl : BOOL;
	bKnock : ARRAY[0..24] OF BOOL;
	bAmmSeqClkP : BOOL;
	AmmSeqValveErr : AmmSequence;
	AmmSeqKnockSigErr : AmmSequence;
	AmmSeqKnockErr : AmmSequence;
	xOpMode : OpMode;
	rOff : REAL; (* individual knock limit offset *)
	rFilt_Fenst1 : ARRAY[0..24] OF REAL; (* used for individual knock limit *)
	rGainFactor : REAL; (* individual knock limit gain factor *)
	rFilterFactor : REAL; (* time constant knock signal filter *)
	iGain_Knck_Intgr_Down : INT := 10;(* scale of knock integrator down for PBC->KLS *)
END_VAR
```

### Program Logical/Knocking/Kn_safi_dmr (IEC) - + knock monitoring with SAFI-DMR

- Kn_safi_dmr.st (not readable text: treated as protected, skipped)

#### Kn_safi_dmr.var - Local variables
```iecst
(********************************************************************
 * COPYRIGHT -- INNIO Company
 ********************************************************************
 * Program: Knck_safi_dmr
 * File: Knck_safi_dmr.var
 * Author: WaldharM
 * Created: October 21, 2011
 ********************************************************************
 * Local variables of program Knck_safi_dmr
 ********************************************************************)
VAR
	AmmSeqKnockErr : AmmSequence;
	bAmmSeqClkP : BOOL;
	bKnock : ARRAY[0..24] OF BOOL;
	TON_SecondTick : TON;
	iCnt_Cyl : USINT;
	ucCylIndex : USINT;
	rCnt_SensorOK : REAL;
	xOpMode : OpMode;
	knCount : ARRAY[0..24] OF UINT;
	knDetected : ARRAY[0..24] OF BOOL;
	rknSumValue : ARRAY[0..24] OF REAL;
	rPr_Knck_Filt : ARRAY[0..24] OF REAL;
	iNum_EngCycCont : UINT;
	iNum_PLC_Cycles : INT;
	iCnt_FiltFreeze : ARRAY[0..24] OF INT;
END_VAR
VAR
	xTOF_SFIKW : ARRAY[0..24] OF TOF;
	BinaryLogicRKS : USINT; (* decision logic for knock system mode  *)
	rKnck_PBC : REAL;
	rInt_Max : REAL;
	rKnck_IP_Red : REAL;
	rKnck_P_Red : REAL;
	rKnck_T2s_Red : REAL;
	rCA_Knck_Red : ARRAY[0..24] OF REAL;
	rInt_Knck_Sum : REAL;
	rInt_Min : REAL;
	rPr_Knck_PBC : REAL;
	rPr_Knck : ARRAY[0..24] OF REAL;
	rInt_MinLim : REAL;
	rInt_MinLim_Raw : REAL;
	rKno_Pmax_Red_EnP : REAL;
	rPmax_Knck_Red : ARRAY[0..24] OF REAL;
	bPmax_Sum_Corr : ARRAY[0..24] OF BOOL;
	rPmax_Knck_Red_Sum : REAL;
	iCnt_Knck_Cyl : USINT;
	bPmax_Freeze : BOOL;
	rPmax_Knck_Red_SumCyl : REAL;
	iCnt_Knck_Cyl_Freeze : USINT;
	bPmax_Freeze_Reset : ARRAY[0..24] OF BOOL;
	xTOF_PmaxReturn : TOF;
	bReset : BOOL;
	bTest_Knck_Error : ARRAY[0..24] OF BOOL;
	bHeavyKnck : BOOL;
	iCnt_Freeze : INT;
	xRamp_Rel_Knck : ARRAY[0..24] OF RAMPE_R;
	iNum_Calc_Adaptiv : INT;
	ssMinIntKlopf : INT;
	rFilterFactor_DMR : REAL;
	rKLmin_DMR : REAL;
	rGainFactor_DMR : REAL;
	rFactOff_DMR : REAL;
	rOff_DMR : REAL;
	rFilt_Pr_Knck : ARRAY[0..24] OF REAL;
	rKLimitVar_DMR : ARRAY[0..24] OF REAL;
END_VAR
```

#### Kn_safe_dmr.fun
```iecst
(********************************************************************
 * COPYRIGHT -- INNIO Company
 ********************************************************************
 * Program: PBC_MFile
 * File: PBC_MFile.fun
 * Author: 502293141
 * Created: October 27, 2014
 ********************************************************************
 * Functions and function blocks of program PBC_MFile
 ********************************************************************)

FUNCTION SCALE : REAL
	VAR_INPUT
		x : REAL;
		x0 : REAL;
		x1 : REAL;
		y0 : REAL;
		y1 : REAL;
	END_VAR
END_FUNCTION

FUNCTION TIME_TO_SEC : REAL (* Returns the Time value in seconds*)
	VAR_INPUT
		in : TIME;
	END_VAR
END_FUNCTION
```

### Program Logical/Knocking/MsgKN (IEC) - + Messages Knocking

- MsgKNCyclic.st (not readable text: treated as protected, skipped)

- MsgKNInit.st (not readable text: treated as protected, skipped)

#### MsgKN.var
```iecst
VAR
	iAdrMM2AmmBase : UDINT;
	iAdrAmmBase2MM : UDINT;
	xMsg3053 : Msg;
	xMsg3054 : Msg;
	xMsg3055 : Msg;
	xMsg3056 : Msg;
	xMsg3057 : Msg;
	xMsg3058 : Msg;
	xMsg3059 : Msg;
	xMsg3060 : Msg;
	xMsg3061 : Msg;
	xMsg3062 : Msg;
	xMsg3063 : Msg;
	xMsg3064 : Msg;
	xMsg3065 : Msg;
	xMsg3066 : Msg;
	xMsg3067 : Msg;
	xMsg3068 : Msg;
	xMsg3069 : Msg;
	xMsg3070 : Msg;
	xMsg3071 : Msg;
	xMsg3072 : Msg;
	xMsg3073 : Msg;
	xMsg3074 : Msg;
	xMsg3075 : Msg;
	xMsg3076 : Msg;
	xMsg3077 : Msg;
	xMsg3078 : Msg;
	xMsg3079 : Msg;
	xMsg3080 : Msg;
	xMsg3081 : Msg;
	xMsg3082 : Msg;
	xMsg3083 : Msg;
	xMsg3084 : Msg;
	xMsg3085 : Msg;
	xMsg3086 : Msg;
	xMsg3087 : Msg;
	xMsg3088 : Msg;
	xMsg3089 : Msg;
	xMsg3090 : Msg;
	xMsg3091 : Msg;
	xMsg3092 : Msg;
	xMsg3279 : Msg;
	xMsg3281 : Msg;
	xMsg3282 : Msg;
	xMsg3339 : Msg;
	xMsg3341 : Msg;
	xMsg3541 : Msg;
	xMsg1081 : Msg;
	xMsg2111 : Msg;
	xMsg2492 : Msg;
	xMsg1048 : Msg;
	xMsg3342 : Msg;
	xOpMode : OpMode;
	xMsg2440 : Msg;
	xMsg2441 : Msg;
END_VAR
```

### Program Logical/Knocking/OUT_Knck (IEC) - + OUT task of knocking modul

- OUT_KnckCyclic.st (not readable text: treated as protected, skipped)

- OUT_KnckInit.st (not readable text: treated as protected, skipped)

#### OUT_Knck.var - Local variables
```iecst
(********************************************************************
 * COPYRIGHT -- INNIO Company
 ********************************************************************
 * Program: OUT_Knck
 * File: OUT_Knck.var
 * Author: WaldharM
 * Created: October 03, 2011
 ********************************************************************
 * Local variables of program OUT_Knck
 ********************************************************************)
VAR
	ucCylinderCount : USINT;
END_VAR
```

### Program Logical/Knocking/VisKN (IEC) - + Visualization task

- VisKNCyclic.st (not readable text: treated as protected, skipped)

- VisKNInit.st (not readable text: treated as protected, skipped)

#### VisKN.var - Local variables
```iecst
(********************************************************************
 * COPYRIGHT -- INNIO Company
 ********************************************************************
 * Program: VisKN
 * File: VisKN.var
 * Author: WaldharM
 * Created: August 13, 2012
 ********************************************************************
 * Local variables of program VisKN
 ********************************************************************)
VAR
	ucCylinderCount : USINT;
	bPBCSensErrInternal : ARRAY[0 .. 24] OF BOOL; (* in-cylinder pressure sensor measuring signal failure  *)
END_VAR
VAR CONSTANT
	GREEN : INT := 229; (*2, 223, 187*)
	RED : INT := 51;
	ORANGE : INT := 48;
	VIOLET : INT := 5;
	BLUE : INT := 11;
	PINK : INT := 18;
	BROWN : INT := 123;
	CYAN : INT := 124;
	YELLOW : INT := 46;
END_VAR
```

### Program Logical/Knocking/ParKN (IEC, version 4.06.0) - + Parameter handling

- perm_par.st (not readable text: treated as protected, skipped)

#### perm_par.var
```iecst
VAR
	tParaIntern : ParaHandler_typ; (*Connector type to perm_par*)
	tMM2ParaBase_ReadBack : MM2ParaBase_type; (*INTERNAL! V4.06 new readback structure for information from previous tasks*)
	bWriteDataObj : BOOL; (* TRUE=write data object module *)
	bDataObjLenErr : BOOL; (*Error occured in permem: data module size missmatch*)
	bCreateDataObj : BOOL; (* TRUE=create new data object *)
	bWriteOnce : BOOL; (* write permanent memory once *)
	DatObjCreate_01 : DatObjCreate; (* data object create *)
	DatObjInfoBak_02 : DatObjInfo; (* data object info *)
	DatObjDelete_01 : DatObjDelete; (* data object delete *)
	DatObjRead_01 : DatObjRead; (* data object read *)
	DatObjRead_02 : DatObjRead; (* manual initiated data object read *)
	DatObjWrite_01 : DatObjWrite; (* data object write *)
	DatObjDelete_02 : DatObjDelete; (* data object delete *)
	DatObjDelete_11 : DatObjDelete; (*Delete Backup File*)
	DatObjInfo_01 : DatObjInfo; (* data object info *)
	DatObjInfo_02 : DatObjInfo; (* data object info *)
	szModuleName : STRING[35]; (* module name of object *)
	szModuleNameBackup : STRING[35]; (* module name of posiibly created backup object *)
	DatObjCopy_01 : DatObjCopy;
	bCopyDataObj : BOOL;
	TON_WarnDelay : TON;
	TON_WritePMEM : TON; (* delay write permanent memory *)
	ulPMPointer : UDINT; (* adress of actual checksum value *)
	ulChecksum : UDINT; (* parameter checksum value *)
	pm_len : UDINT; (* permanent value lenght *)
	ulChecksumOld : UDINT; (* last vlaue of parameter checksum *)
	ulChkValue : UDINT; (* actual value of parameter pointer *)
	pm_id : UDINT; (* permanent value identifier *)
	pm_p : UDINT; (* permanent value pointer *)
	DatObjInfo_META : DatObjInfo;
	DatObjRead_META : DatObjRead;
	szMetaDataRaw : STRING[2000];
	szMetaData : ARRAY[0..4] OF STRING[35];
	szMetaDataVis : ARRAY[0..3] OF STRING[35];
	ssIndex : INT;
	ssCount : INT;
	ucMetaDataRaw : ARRAY[0..2000] OF USINT;
	ssCount2 : INT;
	szMetaDataFile : STRING[10];
	szText1 : STRING[20];
	pv_adr_IN_XX_tPB2MM : UDINT;
	pv_lng : UDINT;
	pv_lng_IN_XX_tPB2MM : UDINT;
	pv_lng_OUT_XX_tPB2MM : UDINT;
	szText2 : STRING[20];
	pv_adr_OUT_XX_tXX2PB : UDINT;
END_VAR
VAR CONSTANT
	ERR_NOERROR : UINT := 0;
END_VAR
VAR
	usPMWriteCnt : UINT;
	pm_Error : UDINT; (* permanent value error *) (* Deleted: pm : ParaMem_typ; permanent memory tags mathias, 22.8.11*)
	fun_Error : UDINT := 0; (*state > 0 = function error*)
	xLocalParaCheck : ParaCheckFUB; (*local function instance to check parameter values*)
	TON_ParaSetupOk : TON;
	bParaCheckSystemOk : BOOL;
	iDebug_ParaOkChecked : UDINT;
	bRestoreBackupDataObj : BOOL := FALSE;
	bRestoreDataObjContent : BOOL := FALSE;
	pm_id_backup : UDINT;
	pm_p_Backup : UDINT;
	DatObjCopy_02 : DatObjCopy;
	bDeleteBackupDataObj : BOOL := FALSE; (*Command to delete backup data module file on purpose*)
	bDebugPara : ARRAY[0..5] OF BOOL;
	ssIndex2 : INT;
	ssIndex3 : INT;
	ssIndex4 : INT;
	ssIndexVis : INT;
	szText : STRING[40];
	pv_adr_Para : UDINT;
	szParaSnippet : ARRAY[0..5] OF STRING[150];
	szParaIndex : STRING[10];
	slValue : DINT;
	iModuleDLD_ResetCount : INT;
	bDownloadDetected : BOOL;
	bFlagParaStructCopyWorking : BOOL; (*true, if cyclic para copying is active, 1 false cycle at every copy *)
	bStoreInitParaInDataObj : BOOL := FALSE;
	bTestflag : BOOL;
	bReadOutMETA_Once : BOOL;
	tParaCheck_iPvAdress : ARRAY[0..5] OF UDINT;
	tParaCheck_iPvLengt : ARRAY[0..5] OF UDINT;
	tParaCheck_rPvValue : ARRAY[0..5] OF REAL;
	tParaCheck_rRangeMIN : ARRAY[0..5] OF REAL;
	tParaCheck_rRangeMAX : ARRAY[0..5] OF REAL;
	tParaCheck_szPvName : ARRAY[0..5] OF STRING[35];
	ssFormatDetected : INT;
	szMetaDataPart : STRING[150];
	szFullTaskName : STRING[35];
	szFullMetaModuleName : STRING[35];
	debugLen : INT;
	debugSize : INT := 0;
	strcat_adr1 : UDINT;
	strcat_adr2 : UDINT;
	ssIndexTN : INT;
	bAlternate : BOOL;
	n : INT;
	iAlternateChecksum : DINT;
	iAlternateChecksumOld : DINT;
	ulDebugChkValue : ARRAY[0..999] OF UDINT;
	Adr1 : UDINT;
	Adr2 : UDINT;
	usPMWriteCntStepsize : UINT := 1; (*different step sizes to help debug*)
	usPMWriteCntXOR : UINT;
	usPMWriteCntAltSum : UINT;
	ulAdrPM : UDINT;
	usChkValuePM : USINT;
	ulAdrPara : UDINT;
	ulPara_len : UDINT;
	usChkValuePara : USINT;
	iDebugCountPMDifferences : DINT := 0;
	bEngineRunDetected : BOOL; (*detection status bit autocommand 100 /101  for engine run state*)
	ucMetaDataDebugInfoLine : ARRAY[0..24] OF STRING[80];
	ssIndexMand : INT := 0;
	szMetaDataMand : STRING[35];
	iMyErrorInfo_Autoreset : DINT; (*internal autoreset counter*)
	ssIndex_Version : INT; (*internal*)
	ssIndex_BU : INT; (*internal*)
	ssIndex_BU2 : INT; (*internal*)
END_VAR
```

### Package Logical/Monic - MO: MONIC

### Data object Logical/Monic/META_MO (Simple) - MODUL META data file

#### META_MO.dat
```
; *******************************************************************************
; AGGR: Module Meta Data (data module)
;
; This code is confidential and proprietary to the INNIO Company.
; It may not be used in any form, or reproduced in any manner, without the express
; written permission of the INNIO Company.
; Copyright, INNIO Company, 2019
;
; Customized modifications: -
; ------------------------
;
; History:
; -------
; V03.99.00.00	06.03.2013	Weitzer		generated for modular software
; V03.99.02.00	29.05.2013	Zengerer	initial dependencies prepared
; V04.00.00.00	30.01.2014	Denk		new version
; V04.00.01.00	21.04.2014	Denk		new version
; V04.00.02.00	22.07.2014	Denk		tIgn_LimitMonitor corrected
; V04.03.00.00	02.11.2015	Zengerer 	MANDATORYMODULE statement
; V04.05.00.00	27.07.2017	Messner		CAN Diagnosis Picture added
; V04.07.00.00	23.01.2019	Zengerer	Distribute Para task with perm messaage handling capability to all modules, no functional change to V4.06
; V04.10.00.00	09.03.2021	Perktold	change of vvm IN_MO.bMisfCOn on source side to cyclic#1 (from 2)
;
; Instructions for use:
; --------------------
; make only changes at the version numbers
;
; Outstandings:
; ------------
;
; *******************************************************************************
;
"<META>"
;
; Module ID
"<MODUL>MO</MODUL>"
;
; Module Version (xx.yy.zz.cc)
"<VERSION>04.10.00.00</VERSION>"
;
; Module Basisupdate Version BU (00-99)
"<BASISUPDATE_VERSION>00</BASISUPDATE_VERSION>"
;
; Optional: specify order number for limitated module usage
"<ORDER></ORDER>" ;<!--(optional for restricted customizations; missing statement makes module valid for all orders)-->
;
; Parameter Check <PARAn Name='aAbcdef' MIN='xxx' MAX='yyy' />  (watch for correct spacings and apostrophs!)
"<PARAMETER_CHK>"
"	<PARA1 Name='iEng_Motortype' MIN='208' MAX='920' />"
"	<PARA2 />"
"	<PARA3 />"
"	<PARA4 />"
"	<PARA5 />"
"</PARAMETER_CHK>"
;
; Statement, if engine operation is also allowed without this module (FALSE) or if this module´s parameter check passing is mandatory (TRUE)
"<MANDATORYMODULE>FALSE</MANDATORYMODULE>"
;
; Permanent Datamodule Filenames<!-- enter filenames for counter and INTERNAL parameter only; filename without extention-->
"<DATAMODULES>" ;<!-- optional; mehrere DATAMODULES erlaubt-->
"	<DATAMODULE>par_MO</DATAMODULE>"
"</DATAMODULES>"
;
; Dependencies Modules (MMxx.yy.zz.cc)
"<DEPENDENCIES>"
"	<DEPENDENCY MODULE='AB' VERSION='04.00.00.00' />"
"	<DEPENDENCY MODULE='PB' VERSION='04.00.00.00' />"
"	<DEPENDENCY MODULE='HA' VERSION='04.00.00.00' />"
"	<DEPENDENCY MODULE='EC' VERSION='04.00.00.00' />"
"   <DEPENDENCY VISVERSION='02.06.00.00' />"			; Dependencies Visualization
"</DEPENDENCIES>"
;
; Module function description
"<MODULEFUNCTION>" ;<!-- short overview documentation of module function; add reference to detailed information, if available-->
"	<General>	"
"	CAN communication to Monic device "
"	</General>	"
""
"	<F1 Name='CAN Communication' LastModified='04.00.00.00'>"
"	Manage and monitor CAN communication to Monic device.	"
"	</F1>"
"	<F2 Name='Parameter sending' LastModified='04.00.00.00'>"
"	 Send parameters and operation values to the device.	"
"	</F2>"
"	<F3 Name='Error handling' LastModified='04.00.00.00'>"
"	 Forward errors from Monic to control system. 	"
"	</F3>"
"	<F4 Name='Voltage measuring' LastModified='04.00.00.00'>"
"	 Read ignition voltage measure values. "
"	</F4>"
"	<F5 Name='Operating mode' LastModified='04.00.00.00'>"
"	 Selection of monic operating mode depending on operation mode of the engine "
"	</F5>"
""
"	<Info>"
"	Update 4.00.01.00: data type _tMonicLimitREAL, task IN_MO, for compatible format with MM SAFI	"
"	Update 4.00.02.00: V4.00.2 17.07.2014	Denk	fix Datatype tIgn_LimitMonitor corrected. //LimitMon[ucCountG].kind	"
"   Update 4.00.05.00: CAN diagnosis picture "
"	</Info>"
""
"	<Customized LastModified='4.0.0.0'>	"
"	- Nothing "
"	</Customized>	"
""
"</MODULEFUNCTION>"
;
"</META>"
```
